	PROC rRUNSide1A200()
           	rTestPosTop;
		TPWrite "Side 1 A";
		MoveJ pSafeS1, vmax, fine, tWeldGun;
		!Code Goes Here
		MoveJ pSafeS181, vmax, fine, tWeldGun;
		SingArea\Wrist;
		MoveJ [[1181.97,1536.60,299.24],[0.0635588,0.517232,-0.779106,0.348462],[0,1,-3,1],[9E+09,9E+09,9E+09,9E+09,9E+09,9E+09]], vmax, z10, tWeldGun;
		MoveL [[1181.96,1536.60,-12.62],[0.0635661,0.517237,-0.779104,0.348458],[0,1,-2,1],[9E+09,9E+09,9E+09,9E+09,9E+09,9E+09]], v1000, z10, tWeldGun;
		ArcLStart [[1181.53,1528.23,-13.21],[0.063566,0.517241,-0.779104,0.348451],[0,1,-2,1],[9E+09,9E+09,9E+09,9E+09,9E+09,9E+09]], v10, seam13, weld13\Weave:=weave1, fine, tWeldGun;
		ArcLEnd [[1204.96,1528.67,-13.35],[0.0635597,0.517241,-0.779099,0.348465],[0,1,-2,1],[9E+09,9E+09,9E+09,9E+09,9E+09,9E+09]], v10, seam13, weld13\Weave:=weave1, fine, tWeldGun;
		MoveL [[1204.64,1537.23,-12.62],[0.0635617,0.517239,-0.7791,0.348464],[0,1,-2,1],[9E+09,9E+09,9E+09,9E+09,9E+09,9E+09]], vmax, z10, tWeldGun;
		MoveL [[863.66,1538.85,77.89],[0.0635666,0.517243,-0.779097,0.348464],[0,1,-2,1],[9E+09,9E+09,9E+09,9E+09,9E+09,9E+09]], vmax, z10, tWeldGun;
		MoveJ [[861.58,1461.21,260.09],[0.14949,-0.376148,-0.839997,-0.361347],[0,1,-1,1],[9E+09,9E+09,9E+09,9E+09,9E+09,9E+09]], vmax, z10, tWeldGun;
		MoveL [[863.23,1471.68,-11.89],[0.149517,-0.37621,-0.839967,-0.361342],[0,1,-1,1],[9E+09,9E+09,9E+09,9E+09,9E+09,9E+09]], v1000, z10, tWeldGun;
		ArcLStart [[868.03,1476.60,-13.62],[0.103036,-0.394927,-0.849321,-0.334768],[0,1,-1,1],[9E+09,9E+09,9E+09,9E+09,9E+09,9E+09]], v10, seam13, weld13\Weave:=weave1, fine, tWeldGun;
		ArcLEnd [[889.84,1476.38,-13.62],[0.103038,-0.394927,-0.849321,-0.334769],[0,1,-1,1],[9E+09,9E+09,9E+09,9E+09,9E+09,9E+09]], v10, seam13, weld13\Weave:=weave1, fine, tWeldGun;
		MoveL [[886.08,1463.03,-7.28],[0.149478,-0.376156,-0.840008,-0.361317],[0,1,-1,1],[9E+09,9E+09,9E+09,9E+09,9E+09,9E+09]], vmax, z10, tWeldGun;
		MoveJ [[863.35,1506.96,224.59],[0.0635605,0.517248,-0.779091,0.348471],[0,1,-2,1],[9E+09,9E+09,9E+09,9E+09,9E+09,9E+09]], vmax, z10, tWeldGun;
		MoveL [[863.21,1535.55,-10.64],[0.0635626,0.51725,-0.779093,0.348463],[0,1,-2,1],[9E+09,9E+09,9E+09,9E+09,9E+09,9E+09]], vmax, z10, tWeldGun;
		ArcLStart [[862.97,1528.60,-12.53],[0.0386315,0.528138,-0.780724,0.331736],[0,1,-2,1],[9E+09,9E+09,9E+09,9E+09,9E+09,9E+09]], v10, seam13, weld13\Weave:=weave1, fine, tWeldGun;
		ArcLEnd [[883.17,1528.60,-12.53],[0.0386327,0.528141,-0.780723,0.331734],[0,1,-2,1],[9E+09,9E+09,9E+09,9E+09,9E+09,9E+09]], v10, seam13, weld13\Weave:=weave1, fine, tWeldGun;
		MoveL [[887.77,1539.90,182.89],[0.0635615,0.517251,-0.779088,0.348474],[0,1,-2,1],[9E+09,9E+09,9E+09,9E+09,9E+09,9E+09]], vmax, z10, tWeldGun;
		MoveJ [[1182.52,1470.34,61.27],[0.149538,-0.376243,-0.839941,-0.361358],[0,1,-1,1],[9E+09,9E+09,9E+09,9E+09,9E+09,9E+09]], vmax, z10, tWeldGun;
		MoveL [[1182.53,1470.34,-13.67],[0.149532,-0.376236,-0.839946,-0.361356],[0,1,-1,1],[9E+09,9E+09,9E+09,9E+09,9E+09,9E+09]], v1000, z10, tWeldGun;
		ArcLStart [[1181.98,1475.51,-14.31],[0.12127,-0.382205,-0.84735,-0.348153],[0,1,-1,1],[9E+09,9E+09,9E+09,9E+09,9E+09,9E+09]], v10, seam13, weld13\Weave:=weave1, fine, tWeldGun;
		ArcLEnd [[1205.98,1475.52,-14.31],[0.121276,-0.382215,-0.847342,-0.348161],[0,1,-1,1],[9E+09,9E+09,9E+09,9E+09,9E+09,9E+09]], v10, seam13, weld13\Weave:=weave1, fine, tWeldGun;
		MoveL [[1202.33,1469.98,-15.09],[0.149549,-0.376274,-0.839922,-0.361365],[0,1,-1,1],[9E+09,9E+09,9E+09,9E+09,9E+09,9E+09]], vmax, z10, tWeldGun;
		MoveL [[1203.94,921.98,77.52],[0.149416,-0.376356,-0.839957,-0.361252],[0,1,-1,1],[9E+09,9E+09,9E+09,9E+09,9E+09,9E+09]], vmax, z10, tWeldGun;
		MoveL [[1203.94,921.99,-12.57],[0.149422,-0.37636,-0.83995,-0.361263],[0,1,-1,1],[9E+09,9E+09,9E+09,9E+09,9E+09,9E+09]], v1000, z10, tWeldGun;
		ArcLStart [[1203.92,927.58,-13.22],[0.10136,-0.39649,-0.845914,-0.341982],[0,1,-1,1],[9E+09,9E+09,9E+09,9E+09,9E+09,9E+09]], v10, seam13, weld13\Weave:=weave1, fine, tWeldGun;
		ArcLEnd [[1182.52,927.58,-13.22],[0.101362,-0.396499,-0.845908,-0.341986],[0,1,-1,1],[9E+09,9E+09,9E+09,9E+09,9E+09,9E+09]], v10, seam13, weld13\Weave:=weave1, fine, tWeldGun;
		MoveL [[1177.78,921.50,-1.65],[0.149422,-0.376364,-0.839949,-0.36126],[0,1,-1,1],[9E+09,9E+09,9E+09,9E+09,9E+09,9E+09]], vmax, z10, tWeldGun;
		MoveL [[883.71,921.14,-1.64],[0.149424,-0.37639,-0.839933,-0.361269],[0,1,0,1],[9E+09,9E+09,9E+09,9E+09,9E+09,9E+09]], vmax, z10, tWeldGun;
		MoveL [[883.71,924.70,-6.65],[0.151492,-0.376355,-0.855909,-0.320669],[0,1,-1,1],[9E+09,9E+09,9E+09,9E+09,9E+09,9E+09]], v1000, z10, tWeldGun;
		ArcLStart [[883.71,929.31,-12.65],[0.151491,-0.376316,-0.85593,-0.320657],[0,1,-1,1],[9E+09,9E+09,9E+09,9E+09,9E+09,9E+09]], v10, seam13, weld13\Weave:=weave1, fine, tWeldGun;
		ArcLEnd [[865.11,929.31,-12.65],[0.151488,-0.376316,-0.855931,-0.320655],[0,1,-1,1],[9E+09,9E+09,9E+09,9E+09,9E+09,9E+09]], v10, seam13, weld13\Weave:=weave1, fine, tWeldGun;
		MoveL [[863.70,926.54,-9.64],[0.149437,-0.376438,-0.8399,-0.361292],[0,0,0,1],[9E+09,9E+09,9E+09,9E+09,9E+09,9E+09]], v100, z10, tWeldGun;
		MoveL [[861.26,919.79,117.88],[0.149443,-0.376442,-0.8399,-0.361285],[0,1,-1,1],[9E+09,9E+09,9E+09,9E+09,9E+09,9E+09]], vmax, z0, tWeldGun;
		MoveJ [[868.17,991.07,127.71],[0.0426372,-0.330552,0.858067,-0.39069],[0,1,-2,1],[9E+09,9E+09,9E+09,9E+09,9E+09,9E+09]], vmax, z0, tWeldGun;
		MoveL [[868.52,984.75,-7.25],[0.0429876,-0.330645,0.857998,-0.390725],[0,0,-2,1],[9E+09,9E+09,9E+09,9E+09,9E+09,9E+09]], v1000, z10, tWeldGun;
		ArcLStart [[865.93,978.35,-9.72],[0.0443365,-0.337733,0.871616,-0.352502],[0,0,-1,1],[9E+09,9E+09,9E+09,9E+09,9E+09,9E+09]], v10, seam13, weld13\Weave:=weave1, fine, tWeldGun;
		ArcLEnd [[890.71,978.29,-9.75],[0.0443001,-0.337695,0.871633,-0.3525],[0,0,-1,1],[9E+09,9E+09,9E+09,9E+09,9E+09,9E+09]], v10, seam13, weld13\Weave:=weave1, fine, tWeldGun;
		MoveL [[889.59,992.71,-6.61],[0.0430178,-0.330607,0.858002,-0.390745],[0,0,-2,1],[9E+09,9E+09,9E+09,9E+09,9E+09,9E+09]], vmax, z10, tWeldGun;
		MoveL [[889.59,992.73,75.52],[0.0430306,-0.330621,0.857997,-0.390743],[0,1,-2,1],[9E+09,9E+09,9E+09,9E+09,9E+09,9E+09]], vmax, z10, tWeldGun;
		MoveL [[1177.66,992.72,75.52],[0.0430182,-0.33062,0.857997,-0.390745],[0,0,-2,1],[9E+09,9E+09,9E+09,9E+09,9E+09,9E+09]], vmax, z10, tWeldGun;
		MoveL [[1185.40,982.49,-9.15],[0.0429596,-0.330615,0.858003,-0.390743],[0,0,-2,1],[9E+09,9E+09,9E+09,9E+09,9E+09,9E+09]], v1000, z10, tWeldGun;
		ArcLStart [[1180.06,977.10,-12.03],[0.0429555,-0.330634,0.857992,-0.390751],[0,0,-2,1],[9E+09,9E+09,9E+09,9E+09,9E+09,9E+09]], v10, seam13, weld13\Weave:=weave1, fine, tWeldGun;
		ArcLEnd [[1208.25,977.44,-12.05],[0.0429485,-0.330644,0.85799,-0.390748],[0,0,-2,1],[9E+09,9E+09,9E+09,9E+09,9E+09,9E+09]], v10, seam13, weld13\Weave:=weave1, fine, tWeldGun;
		MoveL [[1207.94,989.04,-11.16],[0.0429397,-0.330625,0.858002,-0.39074],[0,0,-2,1],[9E+09,9E+09,9E+09,9E+09,9E+09,9E+09]], v1000, z10, tWeldGun;
		MoveL [[1207.95,989.04,392.36],[0.0429563,-0.330627,0.857995,-0.39075],[0,1,-2,1],[9E+09,9E+09,9E+09,9E+09,9E+09,9E+09]], vmax, z10, tWeldGun;
		MoveJ [[194.09,1536.38,108.42],[0.0907205,-0.623393,0.712906,0.308084],[0,-1,0,1],[9E+09,9E+09,9E+09,9E+09,9E+09,9E+09]], vmax, z10, tWeldGun;
		MoveL [[194.09,1534.55,44.51],[0.0907126,-0.623398,0.712901,0.308089],[0,-1,0,1],[9E+09,9E+09,9E+09,9E+09,9E+09,9E+09]], vmax, z10, tWeldGun;
		ArcLStart [[188.67,1534.52,-1.78],[0.0904696,-0.623399,0.71298,0.307975],[0,-1,0,1],[9E+09,9E+09,9E+09,9E+09,9E+09,9E+09]], v20, seam13, weld13\Weave:=weave1, fine, tWeldGun;
		ArcLEnd [[157.07,1534.50,-1.61],[0.0904549,-0.623403,0.712983,0.307965],[0,-1,0,1],[9E+09,9E+09,9E+09,9E+09,9E+09,9E+09]], v20, seam13, weld13\Weave:=weave1, fine, tWeldGun;
		MoveL [[158.09,1532.35,8.43],[0.0907075,-0.623402,0.712898,0.30809],[0,-1,0,1],[9E+09,9E+09,9E+09,9E+09,9E+09,9E+09]], vmax, z10, tWeldGun;
		MoveL [[-123.91,1535.35,12.43],[0.0907124,-0.623396,0.712903,0.308089],[1,0,0,1],[9E+09,9E+09,9E+09,9E+09,9E+09,9E+09]], vmax, z10, tWeldGun;
		ArcLStart [[-128.10,1535.33,-0.77],[0.0907065,-0.623392,0.712906,0.308093],[1,0,0,1],[9E+09,9E+09,9E+09,9E+09,9E+09,9E+09]], v20, seam13, weld13\Weave:=weave1, fine, tWeldGun;
		ArcLEnd [[-161.33,1535.32,-0.76],[0.0907026,-0.623409,0.712891,0.308093],[1,0,0,1],[9E+09,9E+09,9E+09,9E+09,9E+09,9E+09]], v20, seam13, weld13\Weave:=weave1, fine, tWeldGun;
		MoveL [[-158.90,1535.32,931.69],[0.0906389,-0.623348,0.712932,0.308139],[1,-2,1,0],[9E+09,9E+09,9E+09,9E+09,9E+09,9E+09]], vmax, z0, tWeldGun;
		MoveJ [[-173.66,614.72,251.09],[0.128906,0.0495871,0.95885,-0.248055],[1,-1,1,0],[9E+09,9E+09,9E+09,9E+09,9E+09,9E+09]], vmax, z0, tWeldGun;
		MoveL [[-146.66,553.40,15.33],[0.15216,0.0393582,0.96563,-0.207021],[1,-1,1,0],[9E+09,9E+09,9E+09,9E+09,9E+09,9E+09]], vmax, z0, tWeldGun;
		ArcLStart [[-147.88,553.18,1.12],[0.150717,0.044516,0.958032,-0.239748],[1,-1,1,0],[9E+09,9E+09,9E+09,9E+09,9E+09,9E+09]], v20, seam13, weld13\Weave:=weave1, fine, tWeldGun;
		ArcLEnd [[-115.28,553.19,1.13],[0.150723,0.044502,0.958032,-0.239744],[1,-1,1,0],[9E+09,9E+09,9E+09,9E+09,9E+09,9E+09]], v20, seam13, weld13\Weave:=weave1, fine, tWeldGun;
		MoveL [[-113.65,555.41,12.33],[0.152159,0.0393397,0.96563,-0.207027],[1,-1,1,0],[9E+09,9E+09,9E+09,9E+09,9E+09,9E+09]], vmax, z0, tWeldGun;
		MoveL [[171.61,552.68,21.42],[0.152083,0.0394694,0.965633,-0.207041],[1,-1,1,0],[9E+09,9E+09,9E+09,9E+09,9E+09,9E+09]], vmax, z0, tWeldGun;
		ArcLStart [[168.61,552.48,-0.51],[0.15096,0.043697,0.959444,-0.234031],[1,-1,1,0],[9E+09,9E+09,9E+09,9E+09,9E+09,9E+09]], v20, seam13, weld13\Weave:=weave1, fine, tWeldGun;
		ArcLEnd [[200.42,552.49,-0.51],[0.150963,0.0436867,0.959444,-0.23403],[1,-1,1,0],[9E+09,9E+09,9E+09,9E+09,9E+09,9E+09]], v20, seam13, weld13\Weave:=weave1, fine, tWeldGun;
		MoveL [[204.25,552.75,13.91],[0.152145,0.0394344,0.965619,-0.207068],[1,-1,1,0],[9E+09,9E+09,9E+09,9E+09,9E+09,9E+09]], vmax, z0, tWeldGun;
		MoveL [[860.18,549.11,14.83],[0.152112,0.039289,0.965636,-0.207043],[0,-2,1,0],[9E+09,9E+09,9E+09,9E+09,9E+09,9E+09]], vmax, z0, tWeldGun;
		ArcLStart [[862.38,548.31,-2.96],[0.133579,0.0504356,0.95444,-0.262026],[0,-1,1,0],[9E+09,9E+09,9E+09,9E+09,9E+09,9E+09]], v20, seam13, weld13\Weave:=weave1, fine, tWeldGun;
		ArcLEnd [[895.35,548.90,-2.97],[0.133556,0.0504648,0.954436,-0.262046],[0,-2,1,0],[9E+09,9E+09,9E+09,9E+09,9E+09,9E+09]], v20, seam13, weld13\Weave:=weave1, fine, tWeldGun;
		MoveL [[895.37,549.34,9.83],[0.15211,0.0392827,0.965635,-0.207047],[0,-2,1,0],[9E+09,9E+09,9E+09,9E+09,9E+09,9E+09]], vmax, z0, tWeldGun;
		MoveL [[1175.32,546.94,11.83],[0.1496,0.0478929,0.95235,-0.261449],[0,-2,1,0],[9E+09,9E+09,9E+09,9E+09,9E+09,9E+09]], vmax, z0, tWeldGun;
		ArcLStart [[1179.08,546.13,-3.58],[0.119147,0.061512,0.947538,-0.290161],[0,-2,1,0],[9E+09,9E+09,9E+09,9E+09,9E+09,9E+09]], v20, seam13, weld13\Weave:=weave1, fine, tWeldGun;
		ArcLEnd [[1209.46,546.13,-3.60],[0.15155,0.0512739,0.944084,-0.288288],[0,-2,1,0],[9E+09,9E+09,9E+09,9E+09,9E+09,9E+09]], v20, seam13, weld13\Weave:=weave1, fine, tWeldGun;
		MoveL [[1183.76,537.75,320.86],[0.152128,0.0394118,0.965637,-0.207003],[0,-2,1,0],[9E+09,9E+09,9E+09,9E+09,9E+09,9E+09]], vmax, z0, tWeldGun;
		MoveJ [[759.22,820.77,477.02],[0.128857,0.0495447,0.958803,-0.24827],[0,-1,1,0],[9E+09,9E+09,9E+09,9E+09,9E+09,9E+09]], vmax, z0, tWeldGun;
		MoveJ [[-401.88,982.38,420.80],[0.377905,-0.177501,-0.908663,-0.00353082],[1,0,1,0],[9E+09,9E+09,9E+09,9E+09,9E+09,9E+09]], vmax, z0, tWeldGun;
		MoveL [[-401.87,982.37,-5.96],[0.377901,-0.177501,-0.908665,-0.00352363],[1,0,1,0],[9E+09,9E+09,9E+09,9E+09,9E+09,9E+09]], v1000, z0, tWeldGun;
		ArcLStart [[-407.78,982.54,-7.55],[0.377944,-0.177367,-0.908673,-0.00361758],[1,0,1,0],[9E+09,9E+09,9E+09,9E+09,9E+09,9E+09]], v10, seam13, weld13\Weave:=weave1, fine, tWeldGun;
		ArcL [[-407.62,961.97,-9.33],[0.377925,-0.177522,-0.908651,-0.00352087],[1,0,1,0],[9E+09,9E+09,9E+09,9E+09,9E+09,9E+09]], v10, seam13, weld13\Weave:=weave1, z10, tWeldGun;
		ArcLEnd [[-429.63,955.24,-8.57],[0.245864,-0.589236,-0.75089,-0.168871],[1,0,2,0],[9E+09,9E+09,9E+09,9E+09,9E+09,9E+09]], v10, seam13, weld13\Weave:=weave1, fine, tWeldGun;
		MoveL [[-432.47,945.01,-6.78],[0.274937,-0.581449,-0.743579,-0.182803],[1,0,2,0],[9E+09,9E+09,9E+09,9E+09,9E+09,9E+09]], vmax, z0, tWeldGun;
		MoveL [[-432.39,895.03,94.24],[0.274951,-0.581467,-0.743558,-0.182811],[1,0,2,0],[9E+09,9E+09,9E+09,9E+09,9E+09,9E+09]], vmax, z0, tWeldGun;
		MoveL [[-1101.20,895.02,94.24],[0.274939,-0.581469,-0.743563,-0.182805],[1,0,2,0],[9E+09,9E+09,9E+09,9E+09,9E+09,9E+09]], vmax, z0, tWeldGun;
		MoveL [[-1101.70,938.01,-1.40],[0.240452,-0.654006,-0.686015,-0.209388],[1,0,2,0],[9E+09,9E+09,9E+09,9E+09,9E+09,9E+09]], v1000, z0, tWeldGun;
		ArcLStart [[-1101.62,952.01,-7.20],[0.240453,-0.653997,-0.686023,-0.209388],[1,0,2,0],[9E+09,9E+09,9E+09,9E+09,9E+09,9E+09]], v10, seam13, weld13\Weave:=weave1, fine, tWeldGun;
		ArcL [[-1123.02,952.13,-5.59],[0.240455,-0.654006,-0.686013,-0.209388],[1,0,2,0],[9E+09,9E+09,9E+09,9E+09,9E+09,9E+09]], v10, seam13, weld13\Weave:=weave1, z10, tWeldGun;
		ArcLEnd [[-1128.50,976.05,-6.40],[0.0369824,0.922972,0.0835342,0.37387],[1,0,3,0],[9E+09,9E+09,9E+09,9E+09,9E+09,9E+09]], v10, seam13, weld13\Weave:=weave1, fine, tWeldGun;
		MoveL [[-1142.99,977.01,6.44],[0.0501214,0.923455,0.0523108,0.376805],[1,0,3,0],[9E+09,9E+09,9E+09,9E+09,9E+09,9E+09]], vmax, z0, tWeldGun;
		MoveJ [[-1224.84,979.29,303.50],[0.0444685,0.923113,0.0666376,0.376092],[1,0,-1,0],[9E+09,9E+09,9E+09,9E+09,9E+09,9E+09]], vmax, z20, tWeldGun;
		MoveL [[-1192.76,1156.53,-4.42],[0.044443,0.923122,0.0666432,0.376072],[1,0,-1,0],[9E+09,9E+09,9E+09,9E+09,9E+09,9E+09]], v1000, z0, tWeldGun;
		ArcLStart [[-1191.66,1156.15,-2.46],[0.0444485,0.92313,0.0666399,0.376052],[1,0,-1,0],[9E+09,9E+09,9E+09,9E+09,9E+09,9E+09]], v10, seam13, weld13\Weave:=weave1, fine, tWeldGun;
		ArcL [[-1191.78,1180.21,-3.92],[0.0444409,0.923134,0.066615,0.376047],[1,0,-1,0],[9E+09,9E+09,9E+09,9E+09,9E+09,9E+09]], v10, seam13, weld13\Weave:=weave1, z10, tWeldGun;
		ArcLEnd [[-1166.74,1189.82,-5.14],[0.269841,0.674631,-0.631942,0.269645],[1,0,0,0],[9E+09,9E+09,9E+09,9E+09,9E+09,9E+09]], v10, seam13, weld13\Weave:=weave1, fine, tWeldGun;
		MoveL [[-1165.81,1197.81,-4.44],[0.289046,0.665942,-0.622199,0.292988],[1,0,0,0],[9E+09,9E+09,9E+09,9E+09,9E+09,9E+09]], vmax, z0, tWeldGun;
		MoveL [[-1167.37,1197.80,267.48],[0.269054,0.631082,-0.684208,0.247398],[1,-1,0,0],[9E+09,9E+09,9E+09,9E+09,9E+09,9E+09]], vmax, z0, tWeldGun;
		MoveJ [[-491.85,1197.38,267.48],[0.269045,0.631086,-0.684208,0.247399],[1,-1,0,0],[9E+09,9E+09,9E+09,9E+09,9E+09,9E+09]], vmax, z0, tWeldGun;
		MoveL [[-493.75,1206.46,4.64],[0.230361,0.671978,-0.666396,0.226485],[1,-1,0,0],[9E+09,9E+09,9E+09,9E+09,9E+09,9E+09]], v1000, z0, tWeldGun;
		ArcLStart [[-493.89,1194.98,-8.68],[0.230347,0.671983,-0.666395,0.226488],[1,-1,0,0],[9E+09,9E+09,9E+09,9E+09,9E+09,9E+09]], v10, seam13, weld13\Weave:=weave1, fine, tWeldGun;
		ArcL [[-474.80,1194.46,-8.19],[0.230358,0.671985,-0.666393,0.22648],[1,-1,0,0],[9E+09,9E+09,9E+09,9E+09,9E+09,9E+09]], v10, seam13, weld13\Weave:=weave1, z10, tWeldGun;
		ArcLEnd [[-467.21,1164.88,-9.76],[0.384925,0.00804859,-0.922637,-0.0225884],[1,-1,1,0],[9E+09,9E+09,9E+09,9E+09,9E+09,9E+09]], v10, seam13, weld13\Weave:=weave1, fine, tWeldGun;
		MoveL [[-460.21,1166.10,-6.29],[0.384934,0.00803439,-0.922633,-0.0226006],[1,-1,1,0],[9E+09,9E+09,9E+09,9E+09,9E+09,9E+09]], vmax, z5, tWeldGun;
		MoveL [[-460.61,1166.13,158.38],[0.384913,0.00804793,-0.922641,-0.0226089],[1,-1,1,0],[9E+09,9E+09,9E+09,9E+09,9E+09,9E+09]], vmax, z5, tWeldGun;
		MoveJ [[-411.67,714.00,66.77],[0.262804,0.646065,-0.670013,0.254199],[1,-1,0,0],[9E+09,9E+09,9E+09,9E+09,9E+09,9E+09]], vmax, z5, tWeldGun;
		MoveL [[-411.69,717.21,-6.09],[0.256237,0.656032,-0.660062,0.261312],[1,-1,0,0],[9E+09,9E+09,9E+09,9E+09,9E+09,9E+09]], vmax, z5, tWeldGun;
		ArcLStart [[-411.68,712.41,-5.70],[0.256247,0.656027,-0.66006,0.261318],[1,-1,0,0],[9E+09,9E+09,9E+09,9E+09,9E+09,9E+09]], v5, seam13, weld13\Weave:=weave1, fine, tWeldGun;
		ArcLEnd [[-433.47,712.42,-5.71],[0.256245,0.656034,-0.660051,0.261328],[1,-1,0,0],[9E+09,9E+09,9E+09,9E+09,9E+09,9E+09]], v5, seam13, weld13\Weave:=weave1, fine, tWeldGun;
		MoveL [[-433.52,712.50,86.63],[0.256209,0.656106,-0.660016,0.261269],[1,-1,0,0],[9E+09,9E+09,9E+09,9E+09,9E+09,9E+09]], vmax, z5, tWeldGun;
		MoveL [[-1103.37,713.70,123.92],[0.256219,0.656103,-0.660014,0.261271],[1,-1,0,0],[9E+09,9E+09,9E+09,9E+09,9E+09,9E+09]], vmax, z5, tWeldGun;
		MoveL [[-1103.36,713.70,-5.85],[0.25622,0.656101,-0.660014,0.261276],[1,-1,0,0],[9E+09,9E+09,9E+09,9E+09,9E+09,9E+09]], vmax, z5, tWeldGun;
		ArcLStart [[-1100.80,710.80,-5.85],[0.25621,0.656115,-0.660005,0.261274],[1,-1,0,0],[9E+09,9E+09,9E+09,9E+09,9E+09,9E+09]], v5, seam13, weld13\Weave:=weave1, fine, tWeldGun;
		ArcLEnd [[-1124.56,710.81,-5.88],[0.256211,0.6561,-0.660011,0.261294],[1,-1,0,0],[9E+09,9E+09,9E+09,9E+09,9E+09,9E+09]], v5, seam13, weld13\Weave:=weave1, fine, tWeldGun;
		MoveL [[-1124.57,723.78,145.38],[0.256225,0.656093,-0.660015,0.261287],[1,-1,0,0],[9E+09,9E+09,9E+09,9E+09,9E+09,9E+09]], vmax, z5, tWeldGun;
		MoveJ [[-1174.22,1417.20,153.64],[0.288404,-0.63354,-0.657568,-0.288193],[1,-1,-2,0],[9E+09,9E+09,9E+09,9E+09,9E+09,9E+09]], vmax, z5, tWeldGun;
		MoveL [[-1186.57,1426.06,2.31],[0.28839,-0.633552,-0.657559,-0.288201],[1,-1,-2,0],[9E+09,9E+09,9E+09,9E+09,9E+09,9E+09]], vmax, z5, tWeldGun;
		ArcLStart [[-1185.81,1430.45,-4.51],[0.288383,-0.633572,-0.657547,-0.288192],[1,-1,-2,0],[9E+09,9E+09,9E+09,9E+09,9E+09,9E+09]], v5, seam13, weld13\Weave:=weave1, fine, tWeldGun;
		ArcLEnd [[-1165.69,1430.23,-5.50],[0.288385,-0.633579,-0.65754,-0.288189],[1,-1,-2,0],[9E+09,9E+09,9E+09,9E+09,9E+09,9E+09]], v5, seam13, weld13\Weave:=weave1, fine, tWeldGun;
		MoveL [[-1165.69,1421.27,86.72],[0.28839,-0.633573,-0.657541,-0.288197],[1,-1,-2,0],[9E+09,9E+09,9E+09,9E+09,9E+09,9E+09]], vmax, z5, tWeldGun;
		MoveL [[-494.06,1426.01,134.66],[0.280642,-0.634844,-0.656104,-0.296212],[1,-1,-2,0],[9E+09,9E+09,9E+09,9E+09,9E+09,9E+09]], vmax, z5, tWeldGun;
		MoveL [[-494.05,1425.99,-2.61],[0.280635,-0.634843,-0.65611,-0.296207],[1,-1,-2,0],[9E+09,9E+09,9E+09,9E+09,9E+09,9E+09]], vmax, z5, tWeldGun;
		ArcLStart [[-494.25,1431.59,-10.43],[0.280631,-0.634852,-0.656104,-0.296205],[1,-1,-2,0],[9E+09,9E+09,9E+09,9E+09,9E+09,9E+09]], v5, seam13, weld13\Weave:=weave1, fine, tWeldGun;
		ArcLEnd [[-471.85,1431.77,-9.45],[0.280622,-0.634875,-0.656087,-0.296202],[1,-1,-2,0],[9E+09,9E+09,9E+09,9E+09,9E+09,9E+09]], v5, seam13, weld13\Weave:=weave1, fine, tWeldGun;
		MoveL [[-471.84,1418.41,452.48],[0.280608,-0.634847,-0.656147,-0.296143],[1,-1,-2,0],[9E+09,9E+09,9E+09,9E+09,9E+09,9E+09]], vmax, z5, tWeldGun;
		MoveJ pSafeS1, vmax, fine, tWeldGun;
	ENDPROC
	PROC ss_200()
           	rTestPosTop;
		TPWrite "Side 1 A";
		MoveJ pSafeS1, vmax, fine, tWeldGun;
		!Code Goes Here
		MoveJ pSafeS181, vmax, fine, tWeldGun;
		SingArea\Wrist;
		MoveJ [[1181.97,1536.60,299.24],[0.0635588,0.517232,-0.779106,0.348462],[0,1,-3,1],[9E+09,9E+09,9E+09,9E+09,9E+09,9E+09]], vmax, z10, tWeldGun;
		MoveL [[1181.96,1536.60,-12.62],[0.0635661,0.517237,-0.779104,0.348458],[0,1,-2,1],[9E+09,9E+09,9E+09,9E+09,9E+09,9E+09]], v1000, z10, tWeldGun;
		ArcLStart [[1181.53,1529.02,-11.65],[0.0635714,0.517237,-0.779104,0.348457],[0,1,-2,1],[9E+09,9E+09,9E+09,9E+09,9E+09,9E+09]], v10, seam13, weld13\Weave:=weave1, fine, tWeldGun;
		ArcLEnd [[1204.96,1529.87,-10.62],[0.0635614,0.517237,-0.779103,0.348461],[0,1,-2,1],[9E+09,9E+09,9E+09,9E+09,9E+09,9E+09]], v10, seam13, weld13\Weave:=weave1, fine, tWeldGun;
		MoveL [[1204.64,1537.23,-12.62],[0.0635617,0.517239,-0.7791,0.348464],[0,1,-2,1],[9E+09,9E+09,9E+09,9E+09,9E+09,9E+09]], vmax, z10, tWeldGun;
		MoveL [[863.66,1538.85,77.89],[0.0635666,0.517243,-0.779097,0.348464],[0,1,-2,1],[9E+09,9E+09,9E+09,9E+09,9E+09,9E+09]], vmax, z10, tWeldGun;
		MoveJ [[861.58,1461.21,260.09],[0.14949,-0.376148,-0.839997,-0.361347],[0,1,-1,1],[9E+09,9E+09,9E+09,9E+09,9E+09,9E+09]], vmax, z10, tWeldGun;
		MoveL [[863.23,1471.68,-11.89],[0.149517,-0.37621,-0.839967,-0.361342],[0,1,-1,1],[9E+09,9E+09,9E+09,9E+09,9E+09,9E+09]], v1000, z10, tWeldGun;
		ArcLStart [[863.88,1474.96,-12.64],[0.149558,-0.376296,-0.839897,-0.361396],[0,1,-1,1],[9E+09,9E+09,9E+09,9E+09,9E+09,9E+09]], v10, seam13, weld13\Weave:=weave1, fine, tWeldGun;
		ArcLEnd [[887.67,1475.21,-13.25],[0.149548,-0.376266,-0.839942,-0.361327],[0,1,-1,1],[9E+09,9E+09,9E+09,9E+09,9E+09,9E+09]], v10, seam13, weld13\Weave:=weave1, fine, tWeldGun;
		MoveL [[886.08,1463.03,-7.28],[0.149478,-0.376156,-0.840008,-0.361317],[0,1,-1,1],[9E+09,9E+09,9E+09,9E+09,9E+09,9E+09]], vmax, z10, tWeldGun;
		MoveJ [[863.35,1506.96,224.59],[0.0635605,0.517248,-0.779091,0.348471],[0,1,-2,1],[9E+09,9E+09,9E+09,9E+09,9E+09,9E+09]], vmax, z10, tWeldGun;
		MoveL [[863.21,1535.55,-10.64],[0.0635626,0.51725,-0.779093,0.348463],[0,1,-2,1],[9E+09,9E+09,9E+09,9E+09,9E+09,9E+09]], vmax, z10, tWeldGun;
		ArcLStart [[862.98,1531.20,-11.14],[0.0635851,0.517245,-0.779094,0.348464],[0,1,-2,1],[9E+09,9E+09,9E+09,9E+09,9E+09,9E+09]], v10, seam13, weld13\Weave:=weave1, fine, tWeldGun;
		ArcLEnd [[887.38,1530.81,-10.94],[0.0635922,0.517251,-0.779089,0.348465],[0,1,-2,1],[9E+09,9E+09,9E+09,9E+09,9E+09,9E+09]], v10, seam13, weld13\Weave:=weave1, fine, tWeldGun;
		MoveL [[887.77,1539.90,182.89],[0.0635615,0.517251,-0.779088,0.348474],[0,1,-2,1],[9E+09,9E+09,9E+09,9E+09,9E+09,9E+09]], vmax, z10, tWeldGun;
		MoveJ [[1182.52,1470.34,61.27],[0.149538,-0.376243,-0.839941,-0.361358],[0,1,-1,1],[9E+09,9E+09,9E+09,9E+09,9E+09,9E+09]], vmax, z10, tWeldGun;
		MoveL [[1182.53,1470.34,-16.07],[0.149529,-0.376231,-0.83995,-0.361353],[0,1,-1,1],[9E+09,9E+09,9E+09,9E+09,9E+09,9E+09]], v1000, z10, tWeldGun;
		ArcLStart [[1181.99,1475.51,-15.52],[0.149552,-0.376279,-0.83992,-0.361363],[0,1,-1,1],[9E+09,9E+09,9E+09,9E+09,9E+09,9E+09]], v10, seam13, weld13\Weave:=weave1, fine, tWeldGun;
		ArcLEnd [[1204.38,1476.47,-15.60],[0.149569,-0.376356,-0.839878,-0.361375],[0,1,-1,1],[9E+09,9E+09,9E+09,9E+09,9E+09,9E+09]], v10, seam13, weld13\Weave:=weave1, fine, tWeldGun;
		MoveL [[1202.33,1469.98,-15.09],[0.149549,-0.376274,-0.839922,-0.361365],[0,1,-1,1],[9E+09,9E+09,9E+09,9E+09,9E+09,9E+09]], vmax, z10, tWeldGun;
		MoveL [[1203.94,921.98,77.52],[0.149416,-0.376356,-0.839957,-0.361252],[0,1,-1,1],[9E+09,9E+09,9E+09,9E+09,9E+09,9E+09]], vmax, z10, tWeldGun;
		MoveL [[1203.94,921.99,-12.97],[0.149422,-0.376348,-0.839957,-0.361259],[0,1,-1,1],[9E+09,9E+09,9E+09,9E+09,9E+09,9E+09]], v1000, z10, tWeldGun;
		ArcLStart [[1203.94,928.79,-14.21],[0.149423,-0.376362,-0.839952,-0.361256],[0,1,-1,1],[9E+09,9E+09,9E+09,9E+09,9E+09,9E+09]], v10, seam13, weld13\Weave:=weave1, fine, tWeldGun;
		ArcLEnd [[1178.19,928.79,-14.21],[0.149422,-0.376442,-0.839904,-0.361285],[0,1,-1,1],[9E+09,9E+09,9E+09,9E+09,9E+09,9E+09]], v10, seam13, weld13\Weave:=weave1, fine, tWeldGun;
		MoveL [[1177.78,921.50,-1.65],[0.149422,-0.376364,-0.839949,-0.36126],[0,1,-1,1],[9E+09,9E+09,9E+09,9E+09,9E+09,9E+09]], vmax, z10, tWeldGun;
		MoveL [[883.71,921.14,-1.64],[0.149424,-0.37639,-0.839933,-0.361269],[0,1,0,1],[9E+09,9E+09,9E+09,9E+09,9E+09,9E+09]], vmax, z10, tWeldGun;
		MoveL [[883.71,926.93,-12.24],[0.149423,-0.3764,-0.839927,-0.361273],[0,0,0,1],[9E+09,9E+09,9E+09,9E+09,9E+09,9E+09]], v1000, z10, tWeldGun;
		ArcLStart [[885.40,928.75,-13.38],[0.149454,-0.376503,-0.839867,-0.361295],[0,0,0,1],[9E+09,9E+09,9E+09,9E+09,9E+09,9E+09]], v10, seam13, weld13\Weave:=weave1, fine, tWeldGun;
		ArcLEnd [[866.41,928.73,-13.39],[0.149444,-0.376494,-0.839881,-0.361275],[0,0,0,1],[9E+09,9E+09,9E+09,9E+09,9E+09,9E+09]], v10, seam13, weld13\Weave:=weave1, fine, tWeldGun;
		MoveL [[863.70,926.54,-12.25],[0.149435,-0.37642,-0.839913,-0.361282],[0,0,0,1],[9E+09,9E+09,9E+09,9E+09,9E+09,9E+09]], v100, z10, tWeldGun;
		MoveL [[861.26,919.79,117.88],[0.149443,-0.376442,-0.8399,-0.361285],[0,1,-1,1],[9E+09,9E+09,9E+09,9E+09,9E+09,9E+09]], vmax, z0, tWeldGun;
		MoveJ [[868.17,991.07,127.71],[0.0426372,-0.330552,0.858067,-0.39069],[0,1,-2,1],[9E+09,9E+09,9E+09,9E+09,9E+09,9E+09]], vmax, z0, tWeldGun;
		MoveL [[868.52,991.54,-9.45],[0.0429862,-0.330642,0.857997,-0.390729],[0,0,-2,1],[9E+09,9E+09,9E+09,9E+09,9E+09,9E+09]], v1000, z10, tWeldGun;
		ArcLStart [[865.93,978.35,-10.52],[0.0429801,-0.330651,0.857991,-0.390736],[0,0,-2,1],[9E+09,9E+09,9E+09,9E+09,9E+09,9E+09]], v10, seam13, weld13\Weave:=weave1, fine, tWeldGun;
		ArcLEnd [[888.37,978.36,-11.00],[0.0429914,-0.330695,0.857973,-0.390738],[0,0,-2,1],[9E+09,9E+09,9E+09,9E+09,9E+09,9E+09]], v10, seam13, weld13\Weave:=weave1, fine, tWeldGun;
		MoveL [[889.59,992.71,-9.41],[0.0430222,-0.330607,0.858002,-0.390746],[0,0,-2,1],[9E+09,9E+09,9E+09,9E+09,9E+09,9E+09]], vmax, z10, tWeldGun;
		MoveL [[889.59,992.73,75.52],[0.0430306,-0.330621,0.857997,-0.390743],[0,1,-2,1],[9E+09,9E+09,9E+09,9E+09,9E+09,9E+09]], vmax, z10, tWeldGun;
		MoveL [[1177.66,992.72,75.52],[0.0430182,-0.33062,0.857997,-0.390745],[0,0,-2,1],[9E+09,9E+09,9E+09,9E+09,9E+09,9E+09]], vmax, z10, tWeldGun;
		MoveL [[1185.41,992.70,-11.53],[0.0429716,-0.330606,0.858007,-0.390739],[0,0,-2,1],[9E+09,9E+09,9E+09,9E+09,9E+09,9E+09]], v1000, z10, tWeldGun;
		ArcLStart [[1180.66,978.10,-13.63],[0.0429557,-0.330625,0.857997,-0.390747],[0,0,-2,1],[9E+09,9E+09,9E+09,9E+09,9E+09,9E+09]], v10, seam13, weld13\Weave:=weave1, fine, tWeldGun;
		ArcLEnd [[1207.05,977.71,-13.62],[0.0429527,-0.330628,0.857994,-0.390751],[0,0,-2,1],[9E+09,9E+09,9E+09,9E+09,9E+09,9E+09]], v10, seam13, weld13\Weave:=weave1, fine, tWeldGun;
		MoveL [[1207.94,989.04,-11.16],[0.0429397,-0.330625,0.858002,-0.39074],[0,0,-2,1],[9E+09,9E+09,9E+09,9E+09,9E+09,9E+09]], v1000, z10, tWeldGun;
		MoveL [[1207.95,989.04,392.36],[0.0429563,-0.330627,0.857995,-0.39075],[0,1,-2,1],[9E+09,9E+09,9E+09,9E+09,9E+09,9E+09]], vmax, z10, tWeldGun;
		MoveJ [[194.09,1536.38,108.42],[0.0907205,-0.623393,0.712906,0.308084],[0,-1,0,1],[9E+09,9E+09,9E+09,9E+09,9E+09,9E+09]], vmax, z10, tWeldGun;
		MoveL [[194.09,1534.55,44.51],[0.0907126,-0.623398,0.712901,0.308089],[0,-1,0,1],[9E+09,9E+09,9E+09,9E+09,9E+09,9E+09]], vmax, z10, tWeldGun;
		ArcLStart [[191.25,1532.54,0.05],[0.0904838,-0.623408,0.712969,0.30798],[0,-1,0,1],[9E+09,9E+09,9E+09,9E+09,9E+09,9E+09]], v20, seam13, weld13\Weave:=weave1, fine, tWeldGun;
		ArcLEnd [[157.22,1532.54,0.51],[0.090482,-0.623409,0.712967,0.307981],[0,-1,0,1],[9E+09,9E+09,9E+09,9E+09,9E+09,9E+09]], v20, seam13, weld13\Weave:=weave1, fine, tWeldGun;
		MoveL [[158.09,1532.35,8.43],[0.0907075,-0.623402,0.712898,0.30809],[0,-1,0,1],[9E+09,9E+09,9E+09,9E+09,9E+09,9E+09]], vmax, z10, tWeldGun;
		MoveL [[-123.91,1535.35,12.43],[0.0907124,-0.623396,0.712903,0.308089],[1,0,0,1],[9E+09,9E+09,9E+09,9E+09,9E+09,9E+09]], vmax, z10, tWeldGun;
		ArcLStart [[-126.92,1534.33,1.43],[0.0907044,-0.623405,0.712895,0.308091],[1,0,0,1],[9E+09,9E+09,9E+09,9E+09,9E+09,9E+09]], v20, seam13, weld13\Weave:=weave1, fine, tWeldGun;
		ArcLEnd [[-160.92,1534.33,1.44],[0.090708,-0.623403,0.712896,0.308092],[1,0,0,1],[9E+09,9E+09,9E+09,9E+09,9E+09,9E+09]], v20, seam13, weld13\Weave:=weave1, fine, tWeldGun;
		MoveL [[-158.90,1535.32,931.69],[0.0906389,-0.623348,0.712932,0.308139],[1,-2,1,0],[9E+09,9E+09,9E+09,9E+09,9E+09,9E+09]], vmax, z0, tWeldGun;
		MoveJ [[-173.66,614.72,251.09],[0.128906,0.0495871,0.95885,-0.248055],[1,-1,1,0],[9E+09,9E+09,9E+09,9E+09,9E+09,9E+09]], vmax, z0, tWeldGun;
		MoveL [[-146.66,553.40,15.33],[0.15216,0.0393582,0.96563,-0.207021],[1,-1,1,0],[9E+09,9E+09,9E+09,9E+09,9E+09,9E+09]], vmax, z0, tWeldGun;
		ArcLStart [[-146.66,553.39,2.32],[0.152156,0.0393511,0.965628,-0.207036],[1,-1,1,0],[9E+09,9E+09,9E+09,9E+09,9E+09,9E+09]], v20, seam13, weld13\Weave:=weave1, fine, tWeldGun;
		ArcLEnd [[-114.67,554.39,1.31],[0.152148,0.0393507,0.965628,-0.207043],[1,-1,1,0],[9E+09,9E+09,9E+09,9E+09,9E+09,9E+09]], v20, seam13, weld13\Weave:=weave1, fine, tWeldGun;
		MoveL [[-113.65,555.41,12.33],[0.152159,0.0393397,0.96563,-0.207027],[1,-1,1,0],[9E+09,9E+09,9E+09,9E+09,9E+09,9E+09]], vmax, z0, tWeldGun;
		MoveL [[171.61,552.68,21.42],[0.152083,0.0394694,0.965633,-0.207041],[1,-1,1,0],[9E+09,9E+09,9E+09,9E+09,9E+09,9E+09]], vmax, z0, tWeldGun;
		ArcLStart [[171.63,552.69,-0.51],[0.152132,0.0394445,0.96562,-0.207073],[1,-1,1,0],[9E+09,9E+09,9E+09,9E+09,9E+09,9E+09]], v20, seam13, weld13\Weave:=weave1, fine, tWeldGun;
		ArcLEnd [[202.63,552.69,-0.52],[0.152129,0.0394303,0.965618,-0.207083],[1,-1,1,0],[9E+09,9E+09,9E+09,9E+09,9E+09,9E+09]], v20, seam13, weld13\Weave:=weave1, fine, tWeldGun;
		MoveL [[204.25,552.75,13.91],[0.152145,0.0394344,0.965619,-0.207068],[1,-1,1,0],[9E+09,9E+09,9E+09,9E+09,9E+09,9E+09]], vmax, z0, tWeldGun;
		MoveL [[860.18,549.11,14.83],[0.152112,0.039289,0.965636,-0.207043],[0,-2,1,0],[9E+09,9E+09,9E+09,9E+09,9E+09,9E+09]], vmax, z0, tWeldGun;
		ArcLStart [[860.21,550.17,-4.16],[0.152159,0.0392088,0.965632,-0.207039],[0,-2,1,0],[9E+09,9E+09,9E+09,9E+09,9E+09,9E+09]], v20, seam13, weld13\Weave:=weave1, fine, tWeldGun;
		ArcLEnd [[895.96,549.20,-3.18],[0.152141,0.039174,0.965634,-0.207051],[0,-2,1,0],[9E+09,9E+09,9E+09,9E+09,9E+09,9E+09]], v20, seam13, weld13\Weave:=weave1, fine, tWeldGun;
		MoveL [[895.37,549.34,9.83],[0.15211,0.0392827,0.965635,-0.207047],[0,-2,1,0],[9E+09,9E+09,9E+09,9E+09,9E+09,9E+09]], vmax, z0, tWeldGun;
		MoveL [[1175.32,546.94,11.83],[0.1496,0.0478929,0.95235,-0.261449],[0,-2,1,0],[9E+09,9E+09,9E+09,9E+09,9E+09,9E+09]], vmax, z0, tWeldGun;
		ArcLStart [[1177.31,546.94,-3.16],[0.149595,0.0478934,0.95235,-0.261454],[0,-2,1,0],[9E+09,9E+09,9E+09,9E+09,9E+09,9E+09]], v20, seam13, weld13\Weave:=weave1, fine, tWeldGun;
		ArcLEnd [[1209.31,546.95,-3.16],[0.149595,0.0478909,0.95235,-0.261454],[0,-2,1,0],[9E+09,9E+09,9E+09,9E+09,9E+09,9E+09]], v20, seam13, weld13\Weave:=weave1, fine, tWeldGun;
		MoveL [[1183.76,537.75,320.86],[0.152128,0.0394118,0.965637,-0.207003],[0,-2,1,0],[9E+09,9E+09,9E+09,9E+09,9E+09,9E+09]], vmax, z0, tWeldGun;
		MoveJ [[759.22,820.77,477.02],[0.128857,0.0495447,0.958803,-0.24827],[0,-1,1,0],[9E+09,9E+09,9E+09,9E+09,9E+09,9E+09]], vmax, z0, tWeldGun;
		MoveJ [[-401.88,982.38,420.80],[0.377905,-0.177501,-0.908663,-0.00353082],[1,0,1,0],[9E+09,9E+09,9E+09,9E+09,9E+09,9E+09]], vmax, z0, tWeldGun;
		MoveL [[-401.87,982.37,-5.96],[0.377901,-0.177501,-0.908665,-0.00352363],[1,0,1,0],[9E+09,9E+09,9E+09,9E+09,9E+09,9E+09]], v1000, z0, tWeldGun;
		ArcLStart [[-407.18,982.54,-5.95],[0.377941,-0.177364,-0.908675,-0.00361829],[1,0,1,0],[9E+09,9E+09,9E+09,9E+09,9E+09,9E+09]], v10, seam13, weld13\Weave:=weave1, fine, tWeldGun;
		ArcL [[-407.21,961.97,-7.34],[0.377917,-0.177516,-0.908656,-0.00352015],[1,0,1,0],[9E+09,9E+09,9E+09,9E+09,9E+09,9E+09]], v10, seam13, weld13\Weave:=weave1, z10, tWeldGun;
		ArcLEnd [[-429.48,955.83,-6.96],[0.274941,-0.581479,-0.743555,-0.1828],[1,0,2,0],[9E+09,9E+09,9E+09,9E+09,9E+09,9E+09]], v10, seam13, weld13\Weave:=weave1, fine, tWeldGun;
		MoveL [[-432.47,945.01,-6.78],[0.274937,-0.581449,-0.743579,-0.182803],[1,0,2,0],[9E+09,9E+09,9E+09,9E+09,9E+09,9E+09]], vmax, z0, tWeldGun;
		MoveL [[-432.39,895.03,94.24],[0.274951,-0.581467,-0.743558,-0.182811],[1,0,2,0],[9E+09,9E+09,9E+09,9E+09,9E+09,9E+09]], vmax, z0, tWeldGun;
		MoveL [[-1101.20,895.02,94.24],[0.274939,-0.581469,-0.743563,-0.182805],[1,0,2,0],[9E+09,9E+09,9E+09,9E+09,9E+09,9E+09]], vmax, z0, tWeldGun;
		MoveL [[-1101.21,942.37,-3.25],[0.274946,-0.581512,-0.743526,-0.182807],[1,0,2,0],[9E+09,9E+09,9E+09,9E+09,9E+09,9E+09]], v1000, z0, tWeldGun;
		ArcLStart [[-1099.81,952.01,-6.02],[0.23841,-0.593999,-0.734594,-0.225162],[1,0,2,0],[9E+09,9E+09,9E+09,9E+09,9E+09,9E+09]], v10, seam13, weld13\Weave:=weave1, fine, tWeldGun;
		ArcL [[-1121.08,951.80,-5.63],[0.238289,-0.634044,-0.696044,-0.238181],[1,0,2,0],[9E+09,9E+09,9E+09,9E+09,9E+09,9E+09]], v10, seam13, weld13\Weave:=weave1, z10, tWeldGun;
		ArcLEnd [[-1129.28,975.89,-6.00],[0.0369776,0.92297,0.0835389,0.373873],[1,0,3,0],[9E+09,9E+09,9E+09,9E+09,9E+09,9E+09]], v10, seam13, weld13\Weave:=weave1, fine, tWeldGun;
		MoveL [[-1142.99,977.01,6.44],[0.0501214,0.923455,0.0523108,0.376805],[1,0,3,0],[9E+09,9E+09,9E+09,9E+09,9E+09,9E+09]], vmax, z0, tWeldGun;
		MoveJ [[-1142.58,979.31,303.50],[0.0444513,0.923112,0.0666342,0.376096],[1,0,-1,0],[9E+09,9E+09,9E+09,9E+09,9E+09,9E+09]], vmax, z20, tWeldGun;
		MoveL [[-1192.76,1156.53,-4.42],[0.044443,0.923122,0.0666432,0.376072],[1,0,-1,0],[9E+09,9E+09,9E+09,9E+09,9E+09,9E+09]], v1000, z0, tWeldGun;
		ArcLStart [[-1192.23,1155.72,-3.63],[0.0444473,0.923132,0.0666323,0.376048],[1,0,-1,0],[9E+09,9E+09,9E+09,9E+09,9E+09,9E+09]], v10, seam13, weld13\Weave:=weave1, fine, tWeldGun;
		ArcL [[-1191.71,1175.69,-5.33],[0.0444379,0.923126,0.0666324,0.376065],[1,0,-1,0],[9E+09,9E+09,9E+09,9E+09,9E+09,9E+09]], v10, seam13, weld13\Weave:=weave1, z10, tWeldGun;
		ArcLEnd [[-1165.81,1187.00,-4.44],[0.28905,0.665936,-0.622204,0.292989],[1,0,0,0],[9E+09,9E+09,9E+09,9E+09,9E+09,9E+09]], v10, seam13, weld13\Weave:=weave1, fine, tWeldGun;
		MoveL [[-1165.81,1197.81,-4.44],[0.289046,0.665942,-0.622199,0.292988],[1,0,0,0],[9E+09,9E+09,9E+09,9E+09,9E+09,9E+09]], vmax, z0, tWeldGun;
		MoveL [[-1167.37,1197.80,267.48],[0.269054,0.631082,-0.684208,0.247398],[1,-1,0,0],[9E+09,9E+09,9E+09,9E+09,9E+09,9E+09]], vmax, z0, tWeldGun;
		MoveJ [[-491.85,1197.38,267.48],[0.269045,0.631086,-0.684208,0.247399],[1,-1,0,0],[9E+09,9E+09,9E+09,9E+09,9E+09,9E+09]], vmax, z0, tWeldGun;
		MoveL [[-495.49,1197.07,-6.30],[0.260132,0.661057,-0.654909,0.257739],[1,-1,0,0],[9E+09,9E+09,9E+09,9E+09,9E+09,9E+09]], v1000, z0, tWeldGun;
		ArcLStart [[-495.49,1192.07,-6.30],[0.260133,0.661061,-0.654906,0.257736],[1,-1,0,0],[9E+09,9E+09,9E+09,9E+09,9E+09,9E+09]], v10, seam13, weld13\Weave:=weave1, fine, tWeldGun;
		ArcL [[-474.53,1190.57,-6.48],[0.263861,0.655019,-0.660957,0.253897],[1,-1,0,0],[9E+09,9E+09,9E+09,9E+09,9E+09,9E+09]], v10, seam13, weld13\Weave:=weave1, z10, tWeldGun;
		ArcLEnd [[-467.21,1164.88,-8.10],[0.384925,0.00804232,-0.922637,-0.0225898],[1,-1,1,0],[9E+09,9E+09,9E+09,9E+09,9E+09,9E+09]], v10, seam13, weld13\Weave:=weave1, fine, tWeldGun;
		MoveL [[-460.21,1166.10,-6.29],[0.384934,0.00803439,-0.922633,-0.0226006],[1,-1,1,0],[9E+09,9E+09,9E+09,9E+09,9E+09,9E+09]], vmax, z5, tWeldGun;
		MoveL [[-460.61,1166.12,771.55],[0.384916,0.00803537,-0.92264,-0.0226078],[1,-1,1,0],[9E+09,9E+09,9E+09,9E+09,9E+09,9E+09]], vmax, z5, tWeldGun;
		MoveJ pSafeS1, vmax, fine, tWeldGun;
	ENDPROC

	PROC rRUNSIDE1A100()
		MoveJ [[895.91,925.45,959.23],[0.222593,0.0151737,0.948305,-0.225698],[0,-1,0,0],[9E+09,9E+09,9E+09,9E+09,9E+09,9E+09]], vmax, z50, tWeldGun;
		MoveJ [[1169.38,1081.61,325.39],[0.296115,-0.947077,-0.052822,0.112127],[0,-2,0,1],[9E+09,9E+09,9E+09,9E+09,9E+09,9E+09]], vmax, z50, tWeldGun;
		MoveL [[1189.00,1080.17,4.63],[0.333707,-0.921868,0.118398,-0.157423],[0,-2,-1,1],[9E+09,9E+09,9E+09,9E+09,9E+09,9E+09]], v1000, z50, tWeldGun;
		ArcLStart [[1189.77,1081.15,-9.31],[0.333708,-0.921874,0.1184,-0.157385],[0,-2,-1,1],[9E+09,9E+09,9E+09,9E+09,9E+09,9E+09]], v10, seam13, weld13\Weave:=weave1, fine, tWeldGun;
		ArcLEnd [[1155.36,1080.96,-9.32],[0.333709,-0.921872,0.118413,-0.157384],[0,-2,-1,1],[9E+09,9E+09,9E+09,9E+09,9E+09,9E+09]], v10, seam13, weld13\Weave:=weave1, fine, tWeldGun;
		MoveL [[1157.55,1079.96,5.67],[0.333709,-0.921874,0.118398,-0.157383],[0,-2,-1,1],[9E+09,9E+09,9E+09,9E+09,9E+09,9E+09]], vmax, z5, tWeldGun;
		MoveL [[867.14,1075.23,8.88],[0.379709,-0.916742,-0.0425212,0.116612],[0,-2,-1,1],[9E+09,9E+09,9E+09,9E+09,9E+09,9E+09]], vmax, z5, tWeldGun;
		ArcLStart [[867.14,1076.23,-4.29],[0.379693,-0.916748,-0.0425036,0.116619],[0,-2,-1,1],[9E+09,9E+09,9E+09,9E+09,9E+09,9E+09]], v10, seam13, weld13\Weave:=weave1, fine, tWeldGun;
		ArcLEnd [[834.55,1076.01,-3.89],[0.379693,-0.916748,-0.0425149,0.116621],[0,-2,-1,1],[9E+09,9E+09,9E+09,9E+09,9E+09,9E+09]], v10, seam13, weld13\Weave:=weave1, fine, tWeldGun;
		MoveL [[834.56,1075.21,12.06],[0.379682,-0.916754,-0.0425092,0.116603],[0,-2,-1,1],[9E+09,9E+09,9E+09,9E+09,9E+09,9E+09]], vmax, z5, tWeldGun;
		MoveL [[175.01,1076.71,9.09],[0.37968,-0.916766,-0.0425174,0.116513],[0,-2,-1,1],[9E+09,9E+09,9E+09,9E+09,9E+09,9E+09]], vmax, z5, tWeldGun;
		ArcLStart [[175.21,1078.51,-3.72],[0.379675,-0.916769,-0.0425118,0.116508],[0,-2,-1,1],[9E+09,9E+09,9E+09,9E+09,9E+09,9E+09]], v10, seam13, weld13\Weave:=weave1, fine, tWeldGun;
		ArcLEnd [[141.33,1079.10,-3.72],[0.379676,-0.91677,-0.0425113,0.116506],[0,-2,-1,1],[9E+09,9E+09,9E+09,9E+09,9E+09,9E+09]], v10, seam13, weld13\Weave:=weave1, fine, tWeldGun;
		MoveL [[140.80,1076.70,8.09],[0.37968,-0.916765,-0.0425275,0.116517],[0,-2,-1,1],[9E+09,9E+09,9E+09,9E+09,9E+09,9E+09]], vmax, z5, tWeldGun;
		MoveL [[-142.04,1078.78,10.05],[0.379684,-0.916763,-0.0426251,0.116487],[0,-2,-1,1],[9E+09,9E+09,9E+09,9E+09,9E+09,9E+09]], vmax, z5, tWeldGun;
		ArcLStart [[-142.04,1079.38,-3.35],[0.379682,-0.916764,-0.0426296,0.116487],[0,-2,-1,1],[9E+09,9E+09,9E+09,9E+09,9E+09,9E+09]], v10, seam13, weld13\Weave:=weave1, fine, tWeldGun;
		ArcLEnd [[-176.44,1079.18,-3.34],[0.379684,-0.916763,-0.0426122,0.116489],[0,-1,-1,1],[9E+09,9E+09,9E+09,9E+09,9E+09,9E+09]], v10, seam13, weld13\Weave:=weave1, fine, tWeldGun;
		SingArea\Wrist;
		MoveL [[-200.44,1085.42,415.26],[0.379667,-0.916774,-0.042596,0.116465],[0,-2,-1,1],[9E+09,9E+09,9E+09,9E+09,9E+09,9E+09]], vmax, z5, tWeldGun;
		MoveJ [[-173.57,559.75,42.74],[0.145109,0.845875,-0.418866,0.296634],[1,0,-1,0],[9E+09,9E+09,9E+09,9E+09,9E+09,9E+09]], vmax, z5, tWeldGun;
		MoveL [[-169.05,562.52,5.19],[0.145175,0.84585,-0.418945,0.296559],[1,0,-1,0],[9E+09,9E+09,9E+09,9E+09,9E+09,9E+09]], vmax, z5, tWeldGun;
		ArcLStart [[-169.04,560.92,-10.02],[0.145172,0.845851,-0.41894,0.296566],[1,0,-1,0],[9E+09,9E+09,9E+09,9E+09,9E+09,9E+09]], v10, seam13, weld13\Weave:=weave1, fine, tWeldGun;
		ArcLEnd [[-135.88,561.25,-8.17],[0.145137,0.845866,-0.418918,0.296573],[1,0,-1,0],[9E+09,9E+09,9E+09,9E+09,9E+09,9E+09]], v10, seam13, weld13\Weave:=weave1, fine, tWeldGun;
		MoveL [[-136.07,560.62,5.61],[0.145144,0.845861,-0.418915,0.296587],[1,0,-1,0],[9E+09,9E+09,9E+09,9E+09,9E+09,9E+09]], vmax, z5, tWeldGun;
		MoveL [[150.30,559.29,2.38],[0.145275,0.845824,-0.41897,0.296549],[0,0,-1,0],[9E+09,9E+09,9E+09,9E+09,9E+09,9E+09]], vmax, z5, tWeldGun;
		ArcLStart [[149.09,560.10,-11.01],[0.145292,0.845814,-0.419001,0.296528],[0,0,-1,0],[9E+09,9E+09,9E+09,9E+09,9E+09,9E+09]], v10, seam13, weld13\Weave:=weave1, fine, tWeldGun;
		ArcLEnd [[180.89,559.95,-10.61],[0.145283,0.845819,-0.418984,0.29654],[0,0,-1,0],[9E+09,9E+09,9E+09,9E+09,9E+09,9E+09]], v10, seam13, weld13\Weave:=weave1, fine, tWeldGun;
		MoveL [[182.55,560.08,7.18],[0.145153,0.845838,-0.418979,0.296555],[0,0,-1,0],[9E+09,9E+09,9E+09,9E+09,9E+09,9E+09]], vmax, z5, tWeldGun;
		MoveL [[840.66,556.48,0.81],[0.145089,0.845777,-0.419076,0.296625],[0,0,-2,0],[9E+09,9E+09,9E+09,9E+09,9E+09,9E+09]], vmax, z5, tWeldGun;
		ArcLStart [[840.24,557.46,-11.97],[0.145114,0.84576,-0.419121,0.296598],[0,0,-2,0],[9E+09,9E+09,9E+09,9E+09,9E+09,9E+09]], v10, seam13, weld13\Weave:=weave1, fine, tWeldGun;
		ArcLEnd [[872.64,557.26,-12.36],[0.145124,0.845757,-0.419128,0.296591],[0,0,-2,0],[9E+09,9E+09,9E+09,9E+09,9E+09,9E+09]], v10, seam13, weld13\Weave:=weave1, fine, tWeldGun;
		MoveL [[873.71,556.66,3.18],[0.145059,0.845775,-0.419071,0.296652],[0,0,-2,0],[9E+09,9E+09,9E+09,9E+09,9E+09,9E+09]], vmax, z5, tWeldGun;
		MoveL [[1157.38,557.31,-2.39],[0.145019,0.845787,-0.419038,0.296683],[0,0,-2,0],[9E+09,9E+09,9E+09,9E+09,9E+09,9E+09]], vmax, z5, tWeldGun;
		ArcLStart [[1159.14,556.83,-14.78],[0.145041,0.845777,-0.419072,0.296654],[0,0,-2,0],[9E+09,9E+09,9E+09,9E+09,9E+09,9E+09]], v10, seam13, weld13\Weave:=weave1, fine, tWeldGun;
		ArcLEnd [[1191.14,556.43,-14.78],[0.145042,0.845778,-0.41907,0.296654],[0,0,-2,0],[9E+09,9E+09,9E+09,9E+09,9E+09,9E+09]], v10, seam13, weld13\Weave:=weave1, fine, tWeldGun;
		MoveL [[1189.43,560.09,663.81],[0.145007,0.845796,-0.418995,0.296726],[0,0,-2,0],[9E+09,9E+09,9E+09,9E+09,9E+09,9E+09]], vmax, z5, tWeldGun;
		MoveJ [[-229.23,1115.81,554.88],[0.237488,0.691166,-0.628837,0.265431],[1,-1,-4,0],[9E+09,9E+09,9E+09,9E+09,9E+09,9E+09]], vmax, z5, tWeldGun;
		MoveL [[-412.06,717.19,27.71],[0.270403,0.66951,-0.638814,0.265624],[1,0,-4,0],[9E+09,9E+09,9E+09,9E+09,9E+09,9E+09]], vmax, z5, tWeldGun;
		MoveL [[-412.07,716.59,-4.48],[0.270405,0.66951,-0.638815,0.26562],[1,0,-4,0],[9E+09,9E+09,9E+09,9E+09,9E+09,9E+09]], vmax, z5, tWeldGun;
		ArcLStart [[-410.88,712.08,-6.38],[0.270414,0.669517,-0.638809,0.265608],[1,0,-4,0],[9E+09,9E+09,9E+09,9E+09,9E+09,9E+09]], v5, seam13, weld13\Weave:=weave1, fine, tWeldGun;
		ArcLEnd [[-432.89,712.28,-6.37],[0.270423,0.669509,-0.638813,0.265609],[1,0,-4,0],[9E+09,9E+09,9E+09,9E+09,9E+09,9E+09]], v5, seam13, weld13\Weave:=weave1, fine, tWeldGun;
		MoveL [[-435.86,714.19,97.74],[0.270409,0.669504,-0.638821,0.265617],[1,0,-4,0],[9E+09,9E+09,9E+09,9E+09,9E+09,9E+09]], vmax, z5, tWeldGun;
		MoveL [[-1100.50,721.09,94.11],[0.270393,0.669535,-0.638788,0.265635],[1,-1,-4,0],[9E+09,9E+09,9E+09,9E+09,9E+09,9E+09]], vmax, z5, tWeldGun;
		MoveL [[-1101.50,713.37,5.61],[0.270374,0.669541,-0.638766,0.265689],[1,-1,-4,0],[9E+09,9E+09,9E+09,9E+09,9E+09,9E+09]], vmax, z5, tWeldGun;
		ArcLStart [[-1101.59,711.00,-6.35],[0.270404,0.669545,-0.638776,0.265626],[1,-1,-4,0],[9E+09,9E+09,9E+09,9E+09,9E+09,9E+09]], v5, seam13, weld13\Weave:=weave1, fine, tWeldGun;
		ArcLEnd [[-1124.75,711.02,-5.59],[0.270396,0.669535,-0.638784,0.265639],[1,-1,-4,0],[9E+09,9E+09,9E+09,9E+09,9E+09,9E+09]], v5, seam13, weld13\Weave:=weave1, fine, tWeldGun;
		MoveL [[-1124.97,712.38,115.49],[0.270384,0.669531,-0.638781,0.26567],[1,-1,-4,0],[9E+09,9E+09,9E+09,9E+09,9E+09,9E+09]], vmax, z5, tWeldGun;
		MoveJ [[-1119.62,941.62,98.59],[0.263153,-0.665669,-0.65042,-0.254146],[1,0,-2,0],[9E+09,9E+09,9E+09,9E+09,9E+09,9E+09]], vmax, z5, tWeldGun;
		MoveL [[-1103.53,941.47,2.67],[0.263185,-0.665692,-0.650383,-0.254147],[1,0,-2,0],[9E+09,9E+09,9E+09,9E+09,9E+09,9E+09]], vmax, z5, tWeldGun;
		ArcLStart [[-1101.53,952.26,-6.90],[0.245387,-0.665955,-0.67203,-0.211343],[1,0,-2,0],[9E+09,9E+09,9E+09,9E+09,9E+09,9E+09]], v5, seam13, weld13\Weave:=weave1, fine, tWeldGun;
		ArcL [[-1122.43,951.87,-6.14],[0.230872,-0.677147,-0.664308,-0.216486],[1,0,-2,0],[9E+09,9E+09,9E+09,9E+09,9E+09,9E+09]], v5, seam13, weld13\Weave:=weave1, z10, tWeldGun;
		ArcLEnd [[-1127.07,980.82,-7.97],[0.0249196,0.926224,0.00835047,0.376057],[1,0,-1,0],[9E+09,9E+09,9E+09,9E+09,9E+09,9E+09]], v5, seam13, weld13\Weave:=weave1, fine, tWeldGun;
		MoveL [[-1139.22,985.18,63.09],[0.0198475,0.898734,0.00249906,0.438039],[1,-1,-1,0],[9E+09,9E+09,9E+09,9E+09,9E+09,9E+09]], vmax, z5, tWeldGun;
		MoveL [[-1197.13,1157.81,50.93],[0.0198552,0.898739,0.00250141,0.438027],[1,-1,-1,0],[9E+09,9E+09,9E+09,9E+09,9E+09,9E+09]], vmax, z5, tWeldGun;
		MoveL [[-1193.29,1156.64,0.22],[0.0202314,0.914596,0.00160149,0.40386],[1,0,-1,0],[9E+09,9E+09,9E+09,9E+09,9E+09,9E+09]], vmax, z5, tWeldGun;
		ArcLStart [[-1188.51,1160.66,-6.37],[0.0436828,0.938874,-0.0114567,0.341288],[1,0,-1,0],[9E+09,9E+09,9E+09,9E+09,9E+09,9E+09]], v5, seam13, weld13\Weave:=weave1, fine, tWeldGun;
		ArcL [[-1189.05,1179.87,-6.18],[0.0350835,0.946422,-0.0228383,0.320208],[1,0,-1,0],[9E+09,9E+09,9E+09,9E+09,9E+09,9E+09]], v5, seam13, weld13\Weave:=weave1, z10, tWeldGun;
		ArcLEnd [[-1166.55,1190.82,-6.94],[0.234885,0.673237,-0.666707,0.216986],[1,-1,0,0],[9E+09,9E+09,9E+09,9E+09,9E+09,9E+09]], v5, seam13, weld13\Weave:=weave1, fine, tWeldGun;
		MoveL [[-1164.13,1200.44,93.33],[0.251271,0.657126,-0.66952,0.23831],[1,-1,0,0],[9E+09,9E+09,9E+09,9E+09,9E+09,9E+09]], vmax, z5, tWeldGun;
		MoveJ [[-1176.39,1428.24,109.35],[0.303454,-0.641239,-0.63752,-0.300495],[1,-1,2,0],[9E+09,9E+09,9E+09,9E+09,9E+09,9E+09]], vmax, z5, tWeldGun;
		MoveL [[-1186.25,1425.03,14.49],[0.262685,-0.660467,-0.654292,-0.258229],[1,0,2,0],[9E+09,9E+09,9E+09,9E+09,9E+09,9E+09]], vmax, z5, tWeldGun;
		ArcLStart [[-1186.06,1432.23,-6.69],[0.26269,-0.660477,-0.654283,-0.258223],[1,0,2,0],[9E+09,9E+09,9E+09,9E+09,9E+09,9E+09]], v5, seam13, weld13\Weave:=weave1, fine, tWeldGun;
		ArcLEnd [[-1165.11,1431.89,-8.08],[0.262694,-0.66048,-0.654277,-0.258225],[1,0,2,0],[9E+09,9E+09,9E+09,9E+09,9E+09,9E+09]], v5, seam13, weld13\Weave:=weave1, fine, tWeldGun;
		MoveL [[-1165.10,1427.68,74.68],[0.262682,-0.660472,-0.654289,-0.258226],[1,0,2,0],[9E+09,9E+09,9E+09,9E+09,9E+09,9E+09]], vmax, z5, tWeldGun;
		MoveL [[-495.20,1424.53,122.41],[0.28862,-0.64963,-0.643265,-0.284411],[1,-1,2,0],[9E+09,9E+09,9E+09,9E+09,9E+09,9E+09]], vmax, z5, tWeldGun;
		MoveL [[-494.27,1423.22,-1.34],[0.28862,-0.649626,-0.643269,-0.284412],[1,-1,2,0],[9E+09,9E+09,9E+09,9E+09,9E+09,9E+09]], vmax, z5, tWeldGun;
		ArcLStart [[-494.28,1431.62,-11.72],[0.288618,-0.64967,-0.643228,-0.284408],[1,-1,2,0],[9E+09,9E+09,9E+09,9E+09,9E+09,9E+09]], v5, seam13, weld13\Weave:=weave1, fine, tWeldGun;
		ArcLEnd [[-472.28,1431.43,-11.12],[0.288622,-0.649659,-0.643237,-0.284409],[1,-1,2,0],[9E+09,9E+09,9E+09,9E+09,9E+09,9E+09]], v5, seam13, weld13\Weave:=weave1, fine, tWeldGun;
		MoveL [[-474.36,1424.49,125.44],[0.288603,-0.649678,-0.643228,-0.284403],[1,-1,2,0],[9E+09,9E+09,9E+09,9E+09,9E+09,9E+09]], vmax, z5, tWeldGun;
		MoveJ [[-479.04,1241.31,118.19],[0.268582,0.650118,-0.664304,0.252806],[1,-1,0,0],[9E+09,9E+09,9E+09,9E+09,9E+09,9E+09]], vmax, z5, tWeldGun;
		MoveL [[-495.83,1201.80,-1.90],[0.268594,0.650121,-0.6643,0.252797],[1,-1,0,0],[9E+09,9E+09,9E+09,9E+09,9E+09,9E+09]], vmax, z5, tWeldGun;
		ArcLStart [[-493.23,1195.81,-8.08],[0.268589,0.650129,-0.664294,0.252795],[1,-1,0,0],[9E+09,9E+09,9E+09,9E+09,9E+09,9E+09]], v5, seam13, weld13\Weave:=weave1, fine, tWeldGun;
		ArcL [[-475.65,1196.01,-7.47],[0.268596,0.650131,-0.664293,0.252787],[1,-1,0,0],[9E+09,9E+09,9E+09,9E+09,9E+09,9E+09]], v5, seam13, weld13\Weave:=weave1, z10, tWeldGun;
		ArcLEnd [[-468.30,1167.75,-9.67],[0.390504,0.0535497,-0.919043,-0.000178963],[1,-1,1,0],[9E+09,9E+09,9E+09,9E+09,9E+09,9E+09]], v5, seam13, weld13\Weave:=weave1, fine, tWeldGun;
		MoveL [[-435.96,1164.94,59.58],[0.390502,0.0535497,-0.919044,-0.000186584],[1,-1,1,0],[9E+09,9E+09,9E+09,9E+09,9E+09,9E+09]], vmax, z5, tWeldGun;
		MoveL [[-398.53,986.99,7.96],[0.390518,0.0535228,-0.919039,-0.00018247],[1,-1,1,0],[9E+09,9E+09,9E+09,9E+09,9E+09,9E+09]], vmax, z5, tWeldGun;
		ArcLStart [[-407.74,987.37,-7.98],[0.390533,0.0535132,-0.919033,-0.000179522],[1,-1,1,0],[9E+09,9E+09,9E+09,9E+09,9E+09,9E+09]], v20, seam13, weld13\Weave:=weave1, fine, tWeldGun;
		ArcL [[-406.86,967.49,-8.33],[0.390542,0.0535142,-0.919029,-0.000188099],[1,-1,1,0],[9E+09,9E+09,9E+09,9E+09,9E+09,9E+09]], v5, seam13, weld13\Weave:=weave1, z10, tWeldGun;
		ArcLEnd [[-428.10,955.08,-6.46],[0.225047,-0.647546,-0.684631,-0.247627],[1,0,2,0],[9E+09,9E+09,9E+09,9E+09,9E+09,9E+09]], v5, seam13, weld13\Weave:=weave1, fine, tWeldGun;
		MoveL [[-432.86,900.19,113.28],[0.289357,-0.647919,-0.645007,-0.283619],[1,-1,2,0],[9E+09,9E+09,9E+09,9E+09,9E+09,9E+09]], vmax, z5, tWeldGun;
		MoveJ [[276.57,1109.67,795.31],[0.28935,-0.647904,-0.645024,-0.283623],[0,0,1,0],[9E+09,9E+09,9E+09,9E+09,9E+09,9E+09]], vmax, z5, tWeldGun;
	ENDPROC
	PROC ProSkid200()
		MoveJ pSafeS1, vmax, fine, tWeldGun;
		MoveL [[-234.96,1621.92,-8.21],[0.194298,-0.276185,-0.910115,-0.24013],[1,-1,1,0],[9E+09,9E+09,9E+09,9E+09,9E+09,9E+09]], vmax, z50, tWeldGun;
		SingArea\Wrist;
		ArcLStart [[-265.19,1628.57,-38.88],[0.243445,-0.67037,-0.655025,-0.249563],[1,0,2,0],[9E+09,9E+09,9E+09,9E+09,9E+09,9E+09]], v40, seam13, weld13, fine, tWeldGun;
		ArcLEnd [[-257.54,1628.57,-38.88],[0.243445,-0.670369,-0.655025,-0.249565],[1,0,2,0],[9E+09,9E+09,9E+09,9E+09,9E+09,9E+09]], v10, seam13, weld13, fine, tWeldGun;
		MoveL [[-258.35,1618.76,-2.87],[0.243441,-0.670362,-0.655032,-0.24957],[1,0,2,0],[9E+09,9E+09,9E+09,9E+09,9E+09,9E+09]], vmax, z20, tWeldGun;
		MoveJ [[-252.87,717.22,166.31],[0.308554,0.634187,-0.646071,0.291883],[1,0,0,0],[9E+09,9E+09,9E+09,9E+09,9E+09,9E+09]], vmax, z20, tWeldGun;
		SingArea\Wrist;
		MoveL [[-273.06,697.08,-39.01],[0.289422,0.639754,-0.670959,0.238254],[1,0,0,0],[9E+09,9E+09,9E+09,9E+09,9E+09,9E+09]], vmax, z20, tWeldGun;
		ArcLStart [[-273.06,687.07,-45.02],[0.289425,0.639748,-0.670962,0.238258],[1,0,0,0],[9E+09,9E+09,9E+09,9E+09,9E+09,9E+09]], v10, seam13, weld13, fine, tWeldGun;
		ArcLEnd [[-266.46,687.08,-45.02],[0.289425,0.63975,-0.67096,0.238257],[1,0,0,0],[9E+09,9E+09,9E+09,9E+09,9E+09,9E+09]], v10, seam13, weld13, fine, tWeldGun;
		MoveL [[-265.17,697.65,3.08],[0.289425,0.639755,-0.670954,0.238258],[1,0,0,0],[9E+09,9E+09,9E+09,9E+09,9E+09,9E+09]], vmax, z20, tWeldGun;
		MoveJ [[1363.12,672.47,163.81],[0.230647,0.704641,-0.28697,0.606574],[0,-1,-1,0],[9E+09,9E+09,9E+09,9E+09,9E+09,9E+09]], vmax, z20, tWeldGun;
		MoveL [[1363.13,672.48,-59.34],[0.230635,0.704646,-0.28697,0.606573],[0,-1,-1,0],[9E+09,9E+09,9E+09,9E+09,9E+09,9E+09]], vmax, z20, tWeldGun;
		ArcLStart [[1395.10,665.67,-59.36],[0.230647,0.704646,-0.286968,0.606569],[0,-1,-1,0],[9E+09,9E+09,9E+09,9E+09,9E+09,9E+09]], v10, seam13, weld13, fine, tWeldGun;
		ArcLEnd [[1393.21,666.82,-105.76],[0.230653,0.704647,-0.286991,0.606554],[0,-1,-1,0],[9E+09,9E+09,9E+09,9E+09,9E+09,9E+09]], v10, seam13, weld13, fine, tWeldGun;
		MoveL [[1360.51,678.95,-105.76],[0.230657,0.704646,-0.286998,0.60655],[0,-1,-1,0],[9E+09,9E+09,9E+09,9E+09,9E+09,9E+09]], vmax, z20, tWeldGun;
		MoveJ [[1360.48,679.11,200.26],[0.227916,0.703475,-0.290109,0.607465],[0,-1,-1,0],[9E+09,9E+09,9E+09,9E+09,9E+09,9E+09]], vmax, z20, tWeldGun;
		MoveJ [[1372.60,1612.03,89.61],[0.238536,-0.688587,-0.26592,-0.631059],[0,-1,-2,0],[9E+09,9E+09,9E+09,9E+09,9E+09,9E+09]], vmax, z20, tWeldGun;
		MoveL [[1372.62,1612.07,-51.09],[0.238534,-0.68856,-0.265944,-0.631079],[0,-1,-2,0],[9E+09,9E+09,9E+09,9E+09,9E+09,9E+09]], vmax, z20, tWeldGun;
		ArcLStart [[1403.05,1622.70,-51.46],[0.238475,-0.688587,-0.265917,-0.631084],[0,-1,-2,0],[9E+09,9E+09,9E+09,9E+09,9E+09,9E+09]], v10, seam13, weld13, fine, tWeldGun;
		ArcLEnd [[1401.72,1623.96,-98.89],[0.23847,-0.688542,-0.266036,-0.631085],[0,-1,-2,0],[9E+09,9E+09,9E+09,9E+09,9E+09,9E+09]], v10, seam13, weld13, fine, tWeldGun;
		MoveL [[1350.78,1600.25,-98.94],[0.23849,-0.68857,-0.265983,-0.631068],[0,-1,-2,0],[9E+09,9E+09,9E+09,9E+09,9E+09,9E+09]], vmax, z20, tWeldGun;
		MoveL [[1286.32,1556.33,142.30],[0.238485,-0.688572,-0.265997,-0.631063],[0,-1,-2,0],[9E+09,9E+09,9E+09,9E+09,9E+09,9E+09]], vmax, z20, tWeldGun;
		MoveJ [[1024.21,1614.84,123.96],[0.621106,-0.285749,-0.670591,-0.287895],[0,0,0,0],[9E+09,9E+09,9E+09,9E+09,9E+09,9E+09]], vmax, z20, tWeldGun;
		MoveL [[1024.31,1614.97,-44.55],[0.621177,-0.285699,-0.670494,-0.288017],[0,0,0,0],[9E+09,9E+09,9E+09,9E+09,9E+09,9E+09]], vmax, z20, tWeldGun;
		ArcLStart [[986.78,1630.52,-48.85],[0.621168,-0.285689,-0.670501,-0.28803],[0,0,0,0],[9E+09,9E+09,9E+09,9E+09,9E+09,9E+09]], v10, seam13, weld13, fine, tWeldGun;
		ArcLEnd [[989.07,1629.80,-94.04],[0.621174,-0.285677,-0.670503,-0.288024],[0,0,0,0],[9E+09,9E+09,9E+09,9E+09,9E+09,9E+09]], v10, seam13, weld13, fine, tWeldGun;
		MoveL [[1031.38,1620.08,-94.06],[0.621173,-0.285694,-0.670496,-0.288025],[0,0,0,0],[9E+09,9E+09,9E+09,9E+09,9E+09,9E+09]], vmax, z20, tWeldGun;
		MoveL [[1050.77,1575.36,86.67],[0.621174,-0.285691,-0.670496,-0.288026],[0,0,0,0],[9E+09,9E+09,9E+09,9E+09,9E+09,9E+09]], vmax, z20, tWeldGun;
		MoveJ [[1013.51,687.74,143.37],[0.59856,0.318284,-0.67023,0.302017],[0,-1,-1,0],[9E+09,9E+09,9E+09,9E+09,9E+09,9E+09]], vmax, z20, tWeldGun;
		MoveL [[1013.45,687.71,-58.15],[0.598615,0.318227,-0.670196,0.302042],[0,-1,-1,0],[9E+09,9E+09,9E+09,9E+09,9E+09,9E+09]], vmax, z20, tWeldGun;
		ArcLStart [[981.75,669.03,-58.14],[0.598616,0.318216,-0.6702,0.302041],[0,-1,-1,0],[9E+09,9E+09,9E+09,9E+09,9E+09,9E+09]], v10, seam13, weld13, fine, tWeldGun;
		ArcLEnd [[981.75,669.03,-102.94],[0.598614,0.318211,-0.670206,0.302041],[0,-1,-1,0],[9E+09,9E+09,9E+09,9E+09,9E+09,9E+09]], v10, seam13, weld13, fine, tWeldGun;
		MoveL [[1021.06,692.65,-100.54],[0.598619,0.318178,-0.670217,0.30204],[0,-1,-1,0],[9E+09,9E+09,9E+09,9E+09,9E+09,9E+09]], vmax, z20, tWeldGun;
		MoveL [[1021.06,692.65,172.93],[0.598621,0.318175,-0.670218,0.302038],[0,-1,-1,0],[9E+09,9E+09,9E+09,9E+09,9E+09,9E+09]], vmax, z20, tWeldGun;
		MoveJ [[962.66,684.38,264.32],[0.236784,0.681997,-0.2918,0.627429],[0,1,1,1],[9E+09,9E+09,9E+09,9E+09,9E+09,9E+09]], vmax, z20, tWeldGun;
		MoveL [[962.64,684.38,-48.75],[0.236792,0.682002,-0.291815,0.627413],[0,1,1,1],[9E+09,9E+09,9E+09,9E+09,9E+09,9E+09]], vmax, z20, tWeldGun;
		ArcLStart [[980.94,668.93,-48.75],[0.236782,0.682005,-0.291808,0.627418],[0,1,1,1],[9E+09,9E+09,9E+09,9E+09,9E+09,9E+09]], v10, seam13, weld13, fine, tWeldGun;
		ArcLEnd [[980.92,669.75,-104.66],[0.236799,0.682008,-0.291831,0.627396],[0,1,1,1],[9E+09,9E+09,9E+09,9E+09,9E+09,9E+09]], v10, seam13, weld13, fine, tWeldGun;
		MoveL [[948.38,696.75,-105.45],[0.234731,0.68317,-0.291592,0.62702],[0,1,1,1],[9E+09,9E+09,9E+09,9E+09,9E+09,9E+09]], vmax, z20, tWeldGun;
		MoveL [[948.40,696.76,143.62],[0.234722,0.683169,-0.291572,0.627035],[0,1,1,1],[9E+09,9E+09,9E+09,9E+09,9E+09,9E+09]], vmax, z20, tWeldGun;
		MoveJ [[975.43,1612.68,308.57],[0.225877,-0.689512,-0.28382,-0.626896],[0,1,0,1],[9E+09,9E+09,9E+09,9E+09,9E+09,9E+09]], vmax, z20, tWeldGun;
		MoveL [[975.55,1612.35,-40.05],[0.22557,-0.689612,-0.283854,-0.626882],[0,0,1,1],[9E+09,9E+09,9E+09,9E+09,9E+09,9E+09]], vmax, z20, tWeldGun;
		ArcLStart [[989.75,1627.18,-40.10],[0.225683,-0.689679,-0.283801,-0.626791],[0,1,1,1],[9E+09,9E+09,9E+09,9E+09,9E+09,9E+09]], v10, seam13, weld13, fine, tWeldGun;
		ArcLEnd [[988.02,1626.51,-103.36],[0.218861,-0.704472,-0.289009,-0.610159],[0,1,1,1],[9E+09,9E+09,9E+09,9E+09,9E+09,9E+09]], v10, seam13, weld13, fine, tWeldGun;
		MoveL [[969.19,1616.42,-103.36],[0.21886,-0.704489,-0.288978,-0.610154],[0,1,1,1],[9E+09,9E+09,9E+09,9E+09,9E+09,9E+09]], vmax, z20, tWeldGun;
		MoveL [[972.04,1615.87,168.33],[0.225681,-0.689708,-0.283758,-0.62678],[0,1,0,1],[9E+09,9E+09,9E+09,9E+09,9E+09,9E+09]], vmax, z20, tWeldGun;
		MoveJ [[748.32,1594.78,-28.74],[0.231269,-0.620927,-0.702805,-0.258902],[0,1,-1,1],[9E+09,9E+09,9E+09,9E+09,9E+09,9E+09]], vmax, z20, tWeldGun;
		MoveL [[748.32,1618.27,-62.58],[0.231267,-0.620927,-0.702807,-0.258898],[0,1,-1,1],[9E+09,9E+09,9E+09,9E+09,9E+09,9E+09]], vmax, z20, tWeldGun;
		ArcLStart [[748.35,1622.75,-67.83],[0.23126,-0.620915,-0.702812,-0.25892],[0,1,-1,1],[9E+09,9E+09,9E+09,9E+09,9E+09,9E+09]], v10, seam13, weld13, fine, tWeldGun;
		ArcLEnd [[720.93,1622.75,-67.82],[0.231262,-0.620925,-0.702803,-0.258918],[0,1,-1,1],[9E+09,9E+09,9E+09,9E+09,9E+09,9E+09]], v10, seam13, weld13, fine, tWeldGun;
		MoveL [[683.13,1622.94,-67.84],[0.231262,-0.620938,-0.702794,-0.258913],[0,1,-1,1],[9E+09,9E+09,9E+09,9E+09,9E+09,9E+09]], vmax, z20, tWeldGun;
		ArcLStart [[681.00,1622.93,-67.87],[0.231258,-0.62095,-0.702784,-0.258913],[0,1,-1,1],[9E+09,9E+09,9E+09,9E+09,9E+09,9E+09]], v10, seam13, weld13, fine, tWeldGun;
		ArcLEnd [[654.73,1623.14,-67.84],[0.231266,-0.620945,-0.702787,-0.258912],[0,1,-1,1],[9E+09,9E+09,9E+09,9E+09,9E+09,9E+09]], v10, seam13, weld13, fine, tWeldGun;
		MoveL [[654.72,1619.33,-13.30],[0.231269,-0.620959,-0.702776,-0.258903],[0,1,-1,1],[9E+09,9E+09,9E+09,9E+09,9E+09,9E+09]], vmax, z20, tWeldGun;
		MoveJ [[37.05,1622.28,-7.90],[0.231269,-0.620971,-0.702762,-0.258912],[1,1,-1,1],[9E+09,9E+09,9E+09,9E+09,9E+09,9E+09]], vmax, z20, tWeldGun;
		MoveL [[37.06,1622.28,-65.61],[0.231267,-0.620964,-0.702769,-0.258912],[1,1,-1,1],[9E+09,9E+09,9E+09,9E+09,9E+09,9E+09]], vmax, z20, tWeldGun;
		ArcLStart [[37.05,1628.08,-65.61],[0.231271,-0.620973,-0.702759,-0.258914],[1,1,-1,1],[9E+09,9E+09,9E+09,9E+09,9E+09,9E+09]], v10, seam13, weld13, fine, tWeldGun;
		ArcLEnd [[7.65,1628.68,-65.60],[0.231271,-0.620979,-0.702755,-0.258912],[1,1,-1,1],[9E+09,9E+09,9E+09,9E+09,9E+09,9E+09]], v10, seam13, weld13, fine, tWeldGun;
		MoveL [[-27.35,1629.08,-65.60],[0.231271,-0.620982,-0.702752,-0.258911],[1,1,0,1],[9E+09,9E+09,9E+09,9E+09,9E+09,9E+09]], vmax, z20, tWeldGun;
		ArcLStart [[-31.75,1629.08,-65.60],[0.231272,-0.620988,-0.702747,-0.258912],[1,1,0,1],[9E+09,9E+09,9E+09,9E+09,9E+09,9E+09]], v10, seam13, weld13, fine, tWeldGun;
		ArcLEnd [[-60.36,1629.07,-65.63],[0.231269,-0.621009,-0.70273,-0.258909],[1,1,0,1],[9E+09,9E+09,9E+09,9E+09,9E+09,9E+09]], v10, seam13, weld13, fine, tWeldGun;
		MoveL [[-63.19,1451.21,44.92],[0.231265,-0.62101,-0.702733,-0.258902],[1,1,0,1],[9E+09,9E+09,9E+09,9E+09,9E+09,9E+09]], vmax, z20, tWeldGun;
		SingArea\Wrist;
		MoveJ [[-220.42,1456.39,142.20],[0.365991,-0.606888,-0.673424,-0.210328],[1,0,1,0],[9E+09,9E+09,9E+09,9E+09,9E+09,9E+09]], vmax, z20, tWeldGun;
		MoveL [[-219.91,1623.63,-54.86],[0.365978,-0.606856,-0.673457,-0.210339],[1,0,1,0],[9E+09,9E+09,9E+09,9E+09,9E+09,9E+09]], vmax, z20, tWeldGun;
		ArcLStart [[-219.83,1630.03,-63.47],[0.36598,-0.606851,-0.67346,-0.21034],[1,0,1,0],[9E+09,9E+09,9E+09,9E+09,9E+09,9E+09]], v10, seam13, weld13, fine, tWeldGun;
		ArcLEnd [[-233.82,1630.03,-62.87],[0.365977,-0.606844,-0.673467,-0.210341],[1,0,1,0],[9E+09,9E+09,9E+09,9E+09,9E+09,9E+09]], v10, seam13, weld13, fine, tWeldGun;
		MoveL [[-229.83,1622.04,44.03],[0.365923,-0.606933,-0.673436,-0.21028],[1,0,1,0],[9E+09,9E+09,9E+09,9E+09,9E+09,9E+09]], vmax, z20, tWeldGun;
		MoveJ [[-238.42,695.07,107.36],[0.416175,0.412803,-0.798145,0.139133],[1,0,0,0],[9E+09,9E+09,9E+09,9E+09,9E+09,9E+09]], vmax, z20, tWeldGun;
		MoveL [[-238.43,695.09,-59.53],[0.416176,0.412786,-0.798155,0.139122],[1,0,0,0],[9E+09,9E+09,9E+09,9E+09,9E+09,9E+09]], vmax, z20, tWeldGun;
		ArcLStart [[-240.41,687.67,-69.36],[0.416165,0.412798,-0.798152,0.139137],[1,0,0,0],[9E+09,9E+09,9E+09,9E+09,9E+09,9E+09]], v10, seam13, weld13, fine, tWeldGun;
		ArcLEnd [[-225.81,687.67,-69.75],[0.416158,0.41281,-0.798148,0.139143],[1,0,0,0],[9E+09,9E+09,9E+09,9E+09,9E+09,9E+09]], v10, seam13, weld13, fine, tWeldGun;
		MoveL [[-226.30,704.95,-17.45],[0.416163,0.412818,-0.79814,0.139151],[1,0,0,0],[9E+09,9E+09,9E+09,9E+09,9E+09,9E+09]], vmax, z20, tWeldGun;
		MoveJ [[-68.54,708.92,-17.46],[0.33715,0.641758,-0.612556,0.315044],[1,0,-1,0],[9E+09,9E+09,9E+09,9E+09,9E+09,9E+09]], vmax, z20, tWeldGun;
		MoveL [[-69.37,694.59,-61.82],[0.293998,0.661849,-0.635411,0.267907],[1,0,-1,0],[9E+09,9E+09,9E+09,9E+09,9E+09,9E+09]], vmax, z20, tWeldGun;
		ArcLStart [[-69.36,687.96,-70.31],[0.294028,0.661818,-0.635424,0.26792],[1,0,-1,0],[9E+09,9E+09,9E+09,9E+09,9E+09,9E+09]], v10, seam13, weld13, fine, tWeldGun;
		ArcLEnd [[-41.96,687.95,-70.52],[0.29404,0.66181,-0.635427,0.267921],[1,0,-1,0],[9E+09,9E+09,9E+09,9E+09,9E+09,9E+09]], v10, seam13, weld13, fine, tWeldGun;
		MoveL [[-6.97,687.95,-70.51],[0.294043,0.661806,-0.635431,0.267916],[0,0,-1,0],[9E+09,9E+09,9E+09,9E+09,9E+09,9E+09]], vmax, z20, tWeldGun;
		ArcLStart [[-6.96,687.54,-70.52],[0.294045,0.661806,-0.635429,0.267919],[0,0,-1,0],[9E+09,9E+09,9E+09,9E+09,9E+09,9E+09]], v10, seam13, weld13, fine, tWeldGun;
		ArcLEnd [[21.80,686.99,-70.51],[0.294054,0.661794,-0.635442,0.267908],[0,0,-1,0],[9E+09,9E+09,9E+09,9E+09,9E+09,9E+09]], v10, seam13, weld13, fine, tWeldGun;
		MoveL [[21.80,693.66,-56.32],[0.294011,0.661823,-0.635446,0.267875],[0,0,-1,0],[9E+09,9E+09,9E+09,9E+09,9E+09,9E+09]], vmax, z20, tWeldGun;
		MoveL [[644.60,694.09,-38.11],[0.29406,0.661788,-0.635447,0.267906],[0,0,-1,0],[9E+09,9E+09,9E+09,9E+09,9E+09,9E+09]], vmax, z20, tWeldGun;
		ArcLStart [[644.53,682.78,-73.42],[0.294076,0.661755,-0.635493,0.267859],[0,0,-1,0],[9E+09,9E+09,9E+09,9E+09,9E+09,9E+09]], v40, seam13, weld13, fine, tWeldGun;
		ArcLEnd [[667.66,682.46,-73.44],[0.294106,0.661729,-0.635513,0.267845],[0,0,-1,0],[9E+09,9E+09,9E+09,9E+09,9E+09,9E+09]], v10, seam13, weld13, fine, tWeldGun;
		MoveL [[706.98,682.46,-73.44],[0.294117,0.661731,-0.635507,0.267842],[0,0,-1,0],[9E+09,9E+09,9E+09,9E+09,9E+09,9E+09]], vmax, z20, tWeldGun;
		ArcLStart [[706.98,682.46,-73.44],[0.294117,0.66173,-0.635507,0.267841],[0,0,-1,0],[9E+09,9E+09,9E+09,9E+09,9E+09,9E+09]], v10, seam13, weld13, fine, tWeldGun;
		ArcLEnd [[732.78,682.64,-73.45],[0.294116,0.66175,-0.635481,0.267856],[0,0,-1,0],[9E+09,9E+09,9E+09,9E+09,9E+09,9E+09]], v10, seam13, weld13, fine, tWeldGun;
		MoveL [[743.36,710.11,-13.87],[0.294132,0.661743,-0.635486,0.267845],[0,0,-1,0],[9E+09,9E+09,9E+09,9E+09,9E+09,9E+09]], vmax, z20, tWeldGun;
		MoveJ [[766.73,689.09,12.78],[0.426939,0.266425,-0.809663,0.301972],[0,-1,0,0],[9E+09,9E+09,9E+09,9E+09,9E+09,9E+09]], vmax, z20, tWeldGun;
		MoveL [[766.72,689.01,-73.04],[0.426946,0.266425,-0.809635,0.302037],[0,-1,0,0],[9E+09,9E+09,9E+09,9E+09,9E+09,9E+09]], vmax, z20, tWeldGun;
		ArcLStart [[753.37,674.21,-83.82],[0.426978,0.266403,-0.80963,0.302027],[0,-1,0,0],[9E+09,9E+09,9E+09,9E+09,9E+09,9E+09]], v10, seam13, weld13, fine, tWeldGun;
		ArcLEnd [[753.94,674.20,-111.42],[0.427004,0.266403,-0.809617,0.302024],[0,-1,0,0],[9E+09,9E+09,9E+09,9E+09,9E+09,9E+09]], v10, seam13, weld13, fine, tWeldGun;
		MoveL [[767.24,687.28,-25.85],[0.427002,0.266345,-0.809691,0.301878],[0,-1,0,0],[9E+09,9E+09,9E+09,9E+09,9E+09,9E+09]], vmax, z20, tWeldGun;
		MoveJ [[43.23,696.82,-1.72],[0.42676,0.266354,-0.810055,0.301235],[0,-1,0,0],[9E+09,9E+09,9E+09,9E+09,9E+09,9E+09]], vmax, z20, tWeldGun;
		MoveL [[42.01,683.49,-78.40],[0.427024,0.26632,-0.809694,0.301862],[0,-1,0,0],[9E+09,9E+09,9E+09,9E+09,9E+09,9E+09]], vmax, z20, tWeldGun;
		ArcLStart [[38.82,680.87,-78.40],[0.427033,0.266358,-0.80967,0.301881],[0,-1,0,0],[9E+09,9E+09,9E+09,9E+09,9E+09,9E+09]], v10, seam13, weld13, fine, tWeldGun;
		ArcLEnd [[40.20,680.75,-109.60],[0.427039,0.266382,-0.80967,0.301849],[0,-1,0,0],[9E+09,9E+09,9E+09,9E+09,9E+09,9E+09]], v10, seam13, weld13, fine, tWeldGun;
		MoveL [[56.60,714.15,-11.47],[0.427063,0.266301,-0.809685,0.301848],[0,-1,0,0],[9E+09,9E+09,9E+09,9E+09,9E+09,9E+09]], vmax, z20, tWeldGun;
		MoveJ [[-90.85,716.79,14.15],[0.243321,0.796043,-0.267285,0.485459],[1,-1,-1,0],[9E+09,9E+09,9E+09,9E+09,9E+09,9E+09]], vmax, z20, tWeldGun;
		MoveL [[-92.64,686.16,-78.85],[0.243349,0.796017,-0.267252,0.485505],[1,-1,-1,0],[9E+09,9E+09,9E+09,9E+09,9E+09,9E+09]], vmax, z20, tWeldGun;
		ArcLStart [[-85.54,680.97,-78.85],[0.243338,0.796021,-0.267256,0.485502],[1,-1,-1,0],[9E+09,9E+09,9E+09,9E+09,9E+09,9E+09]], v10, seam13, weld13, fine, tWeldGun;
		ArcLEnd [[-85.54,680.97,-106.06],[0.243338,0.796019,-0.267253,0.485507],[1,-1,-1,0],[9E+09,9E+09,9E+09,9E+09,9E+09,9E+09]], v10, seam13, weld13, fine, tWeldGun;
		MoveL [[-99.62,700.82,-3.32],[0.243332,0.796035,-0.267233,0.485495],[1,-1,-1,0],[9E+09,9E+09,9E+09,9E+09,9E+09,9E+09]], vmax, z20, tWeldGun;
		MoveJ [[622.81,695.86,-3.35],[0.24331,0.796057,-0.26719,0.485493],[0,-1,-1,0],[9E+09,9E+09,9E+09,9E+09,9E+09,9E+09]], vmax, z20, tWeldGun;
		MoveL [[622.81,678.68,-81.59],[0.243312,0.796055,-0.267198,0.485492],[0,-1,-1,0],[9E+09,9E+09,9E+09,9E+09,9E+09,9E+09]], vmax, z20, tWeldGun;
		ArcLStart [[627.79,674.24,-83.40],[0.243343,0.796045,-0.267192,0.485495],[0,-1,-1,0],[9E+09,9E+09,9E+09,9E+09,9E+09,9E+09]], v10, seam13, weld13, fine, tWeldGun;
		ArcLEnd [[626.78,674.63,-109.81],[0.243358,0.796042,-0.267204,0.485485],[0,-1,-1,0],[9E+09,9E+09,9E+09,9E+09,9E+09,9E+09]], v10, seam13, weld13, fine, tWeldGun;
		MoveL [[610.77,692.21,49.90],[0.243321,0.79605,-0.267267,0.485457],[0,-1,-1,0],[9E+09,9E+09,9E+09,9E+09,9E+09,9E+09]], vmax, z20, tWeldGun;
		MoveJ [[622.12,1614.25,159.14],[0.192579,-0.77773,-0.32949,-0.499486],[0,1,0,1],[9E+09,9E+09,9E+09,9E+09,9E+09,9E+09]], vmax, z20, tWeldGun;
		MoveL [[622.15,1614.23,-75.01],[0.192557,-0.777696,-0.329551,-0.499508],[0,1,0,1],[9E+09,9E+09,9E+09,9E+09,9E+09,9E+09]], vmax, z20, tWeldGun;
		ArcLStart [[640.60,1627.79,-79.81],[0.192567,-0.777665,-0.329604,-0.499517],[0,1,0,1],[9E+09,9E+09,9E+09,9E+09,9E+09,9E+09]], v10, seam13, weld13, fine, tWeldGun;
		ArcLEnd [[640.40,1627.75,-105.01],[0.19256,-0.777691,-0.32956,-0.499508],[0,1,0,1],[9E+09,9E+09,9E+09,9E+09,9E+09,9E+09]], v10, seam13, weld13, fine, tWeldGun;
		MoveL [[622.01,1617.53,-16.15],[0.192549,-0.777705,-0.329542,-0.499501],[0,1,0,1],[9E+09,9E+09,9E+09,9E+09,9E+09,9E+09]], vmax, z20, tWeldGun;
		MoveJ [[-74.83,1621.54,-16.16],[0.19255,-0.777728,-0.329501,-0.499493],[1,1,0,1],[9E+09,9E+09,9E+09,9E+09,9E+09,9E+09]], vmax, z20, tWeldGun;
		MoveL [[-74.84,1632.22,-76.43],[0.192546,-0.777738,-0.329487,-0.499489],[1,1,0,1],[9E+09,9E+09,9E+09,9E+09,9E+09,9E+09]], vmax, z20, tWeldGun;
		ArcLStart [[-72.04,1634.00,-74.85],[0.192535,-0.777754,-0.329462,-0.499484],[1,1,0,1],[9E+09,9E+09,9E+09,9E+09,9E+09,9E+09]], v10, seam13, weld13, fine, tWeldGun;
		ArcLEnd [[-72.05,1633.99,-104.27],[0.19253,-0.777762,-0.329453,-0.49948],[1,1,0,1],[9E+09,9E+09,9E+09,9E+09,9E+09,9E+09]], v10, seam13, weld13, fine, tWeldGun;
		MoveL [[-101.85,1558.57,140.36],[0.192608,-0.777808,-0.329372,-0.499431],[1,1,0,1],[9E+09,9E+09,9E+09,9E+09,9E+09,9E+09]], vmax, z20, tWeldGun;
		MoveJ [[102.30,1319.34,116.73],[0.326866,-0.251271,-0.905673,-0.0988914],[0,-1,1,0],[9E+09,9E+09,9E+09,9E+09,9E+09,9E+09]], vmax, z20, tWeldGun;
		MoveL [[56.99,1626.55,-72.67],[0.410474,-0.275782,-0.84185,-0.216205],[0,0,1,0],[9E+09,9E+09,9E+09,9E+09,9E+09,9E+09]], vmax, z20, tWeldGun;
		ArcLStart [[49.28,1632.40,-74.45],[0.41046,-0.275749,-0.841871,-0.216193],[0,0,1,0],[9E+09,9E+09,9E+09,9E+09,9E+09,9E+09]], v10, seam13, weld13, fine, tWeldGun;
		ArcLEnd [[51.27,1632.00,-107.06],[0.410475,-0.275775,-0.841856,-0.216189],[0,0,1,0],[9E+09,9E+09,9E+09,9E+09,9E+09,9E+09]], v10, seam13, weld13, fine, tWeldGun;
		MoveL [[63.32,1618.59,53.83],[0.41045,-0.275792,-0.841833,-0.216304],[0,0,1,0],[9E+09,9E+09,9E+09,9E+09,9E+09,9E+09]], vmax, z20, tWeldGun;
		MoveJ [[774.48,1618.06,-14.91],[0.410442,-0.275748,-0.841846,-0.216328],[0,0,1,0],[9E+09,9E+09,9E+09,9E+09,9E+09,9E+09]], vmax, z20, tWeldGun;
		MoveL [[774.44,1618.01,-79.45],[0.410464,-0.275799,-0.841828,-0.216288],[0,0,0,0],[9E+09,9E+09,9E+09,9E+09,9E+09,9E+09]], vmax, z20, tWeldGun;
		ArcLStart [[760.64,1625.90,-79.46],[0.410464,-0.275804,-0.841826,-0.216291],[0,0,1,0],[9E+09,9E+09,9E+09,9E+09,9E+09,9E+09]], v10, seam13, weld13, fine, tWeldGun;
		ArcLEnd [[761.81,1625.90,-106.65],[0.410464,-0.2758,-0.841828,-0.216289],[0,0,1,0],[9E+09,9E+09,9E+09,9E+09,9E+09,9E+09]], v10, seam13, weld13, fine, tWeldGun;
		MoveL [[783.26,1604.44,251.05],[0.410482,-0.275804,-0.84182,-0.216279],[0,0,1,0],[9E+09,9E+09,9E+09,9E+09,9E+09,9E+09]], vmax, z20, tWeldGun;
		MoveJ pSafeS1, vmax, fine, tWeldGun;
	ENDPROC
	PROC ProSkid50()
		MoveJ [[314.39,1632.04,274.09],[0.410833,-0.611914,-0.675728,-0.0129978],[0,0,-3,0],[9E+09,9E+09,9E+09,9E+09,9E+09,9E+09]], vmax, z50, tWeldGun;
		MoveL [[314.32,1632.00,-25.30],[0.410826,-0.611972,-0.675681,-0.0129369],[0,0,-3,0],[9E+09,9E+09,9E+09,9E+09,9E+09,9E+09]], vmax, z50, tWeldGun;
		ArcLStart [[314.43,1633.11,-39.30],[0.349657,-0.639186,-0.683585,-0.0435139],[0,0,-3,0],[9E+09,9E+09,9E+09,9E+09,9E+09,9E+09]], v10, seam13, weld13, fine, tWeldGun;
		ArcL [[333.87,1632.50,-40.55],[0.349642,-0.639186,-0.683593,-0.0435083],[0,0,-3,0],[9E+09,9E+09,9E+09,9E+09,9E+09,9E+09]], v10, seam13, weld13, z5, tWeldGun;
		ArcL [[341.01,1631.27,-66.17],[0.317739,-0.654055,-0.683899,-0.0594762],[0,0,-3,0],[9E+09,9E+09,9E+09,9E+09,9E+09,9E+09]], v10, seam13, weld13, z5, tWeldGun;
		ArcLEnd [[358.67,1633.28,-65.92],[0.326244,-0.656849,-0.673963,-0.0888224],[0,0,-3,0],[9E+09,9E+09,9E+09,9E+09,9E+09,9E+09]], v10, seam13, weld13, fine, tWeldGun;
		MoveL [[364.49,1617.70,-14.89],[0.410824,-0.611946,-0.675708,-0.012893],[0,0,-3,0],[9E+09,9E+09,9E+09,9E+09,9E+09,9E+09]], vmax, z50, tWeldGun;
		MoveJ [[320.64,789.47,304.99],[0.235374,0.107276,-0.920325,0.293418],[0,-1,-4,0],[9E+09,9E+09,9E+09,9E+09,9E+09,9E+09]], vmax, z50, tWeldGun;
		MoveL [[320.65,680.04,-28.04],[0.235364,0.107285,-0.920324,0.293424],[0,-1,-4,0],[9E+09,9E+09,9E+09,9E+09,9E+09,9E+09]], vmax, z50, tWeldGun;
		ArcLStart [[320.49,676.84,-46.47],[0.235331,0.107401,-0.920274,0.293565],[0,-1,-4,0],[9E+09,9E+09,9E+09,9E+09,9E+09,9E+09]], v10, seam13, weld13, fine, tWeldGun;
		ArcL [[339.64,676.63,-48.64],[0.235361,0.107405,-0.920265,0.293567],[0,-1,-4,0],[9E+09,9E+09,9E+09,9E+09,9E+09,9E+09]], v5, seam13, weld13, z5, tWeldGun;
		ArcL [[342.53,676.66,-71.41],[0.281426,0.0897427,-0.912937,0.281589],[0,-1,-4,0],[9E+09,9E+09,9E+09,9E+09,9E+09,9E+09]], v5, seam13, weld13, z5, tWeldGun;
		ArcLEnd [[360.55,681.94,-73.50],[0.314989,0.316109,-0.866408,0.224044],[0,-1,-4,0],[9E+09,9E+09,9E+09,9E+09,9E+09,9E+09]], v10, seam13, weld13, fine, tWeldGun;
		MoveL [[365.60,682.37,3.04],[0.235347,0.107379,-0.920294,0.293497],[0,-1,-4,0],[9E+09,9E+09,9E+09,9E+09,9E+09,9E+09]], vmax, z50, tWeldGun;
		MoveJ [[836.02,763.37,35.73],[0.0217026,-0.41169,0.816455,-0.40428],[0,-2,-4,0],[9E+09,9E+09,9E+09,9E+09,9E+09,9E+09]], vmax, z50, tWeldGun;
		MoveL [[856.70,689.76,-27.01],[0.0217072,-0.411704,0.816444,-0.404287],[0,-2,-3,0],[9E+09,9E+09,9E+09,9E+09,9E+09,9E+09]], vmax, z50, tWeldGun;
		ArcLStart [[857.91,678.67,-44.98],[0.0203271,-0.414175,0.82252,-0.389238],[0,-2,-3,0],[9E+09,9E+09,9E+09,9E+09,9E+09,9E+09]], v10, seam13, weld13, fine, tWeldGun;
		ArcL [[836.15,679.48,-46.99],[0.0203132,-0.414191,0.822508,-0.389249],[0,-2,-3,0],[9E+09,9E+09,9E+09,9E+09,9E+09,9E+09]], v10, seam13, weld13, z5, tWeldGun;
		ArcL [[831.91,680.96,-69.65],[0.0726329,-0.437948,0.812132,-0.37864],[0,-2,-3,0],[9E+09,9E+09,9E+09,9E+09,9E+09,9E+09]], v10, seam13, weld13, z5, tWeldGun;
		ArcLEnd [[814.71,680.94,-69.65],[0.0726252,-0.437942,0.812135,-0.378643],[0,-2,-3,0],[9E+09,9E+09,9E+09,9E+09,9E+09,9E+09]], v10, seam13, weld13, fine, tWeldGun;
		MoveL [[809.35,725.26,127.04],[0.0216773,-0.411756,0.816405,-0.404315],[0,-2,-4,0],[9E+09,9E+09,9E+09,9E+09,9E+09,9E+09]], vmax, z50, tWeldGun;
		MoveJ [[841.70,1629.86,72.25],[0.220866,-0.864976,-0.348476,-0.285657],[0,0,-2,0],[9E+09,9E+09,9E+09,9E+09,9E+09,9E+09]], vmax, z50, tWeldGun;
		MoveL [[841.69,1629.87,-34.30],[0.220872,-0.864976,-0.348474,-0.285654],[0,0,-2,0],[9E+09,9E+09,9E+09,9E+09,9E+09,9E+09]], vmax, z50, tWeldGun;
		ArcLStart [[848.66,1634.80,-44.07],[0.220862,-0.865006,-0.348435,-0.28562],[0,0,-2,0],[9E+09,9E+09,9E+09,9E+09,9E+09,9E+09]], v20, seam13, weld13, fine, tWeldGun;
		ArcL [[827.08,1634.97,-46.50],[0.220852,-0.865009,-0.348428,-0.285626],[0,0,-2,0],[9E+09,9E+09,9E+09,9E+09,9E+09,9E+09]], v10, seam13, weld13, z1, tWeldGun;
		ArcL [[824.68,1632.91,-69.83],[0.143373,-0.869884,-0.317855,-0.348876],[0,0,-2,0],[9E+09,9E+09,9E+09,9E+09,9E+09,9E+09]], v10, seam13, weld13, z1, tWeldGun;
		ArcLEnd [[803.26,1635.12,-68.75],[0.265625,-0.855119,-0.383795,-0.225647],[0,0,-3,0],[9E+09,9E+09,9E+09,9E+09,9E+09,9E+09]], v10, seam13, weld13, fine, tWeldGun;
		MoveL [[798.38,1604.44,59.29],[0.220844,-0.86502,-0.348413,-0.285617],[0,0,-2,0],[9E+09,9E+09,9E+09,9E+09,9E+09,9E+09]], vmax, z50, tWeldGun;
		MoveJ [[1012.25,1627.55,26.24],[0.148022,-0.852995,-0.305302,-0.396586],[0,-1,-2,0],[9E+09,9E+09,9E+09,9E+09,9E+09,9E+09]], vmax, z50, tWeldGun;
		MoveL [[1012.25,1627.54,-29.96],[0.148013,-0.852994,-0.305304,-0.39659],[0,-1,-2,0],[9E+09,9E+09,9E+09,9E+09,9E+09,9E+09]], vmax, z50, tWeldGun;
		ArcLStart [[1020.33,1635.81,-42.74],[0.234694,-0.797645,-0.305793,-0.463867],[0,0,-2,0],[9E+09,9E+09,9E+09,9E+09,9E+09,9E+09]], v10, seam13, weld13, fine, tWeldGun;
		ArcLEnd [[1020.32,1636.60,-101.76],[0.234691,-0.797653,-0.305783,-0.463861],[0,0,-2,0],[9E+09,9E+09,9E+09,9E+09,9E+09,9E+09]], v10, seam13, weld13, fine, tWeldGun;
		MoveL [[1000.64,1624.71,1.80],[0.147993,-0.85301,-0.305288,-0.396575],[0,-1,-2,0],[9E+09,9E+09,9E+09,9E+09,9E+09,9E+09]], vmax, z50, tWeldGun;
		MoveJ [[999.85,699.71,74.25],[0.145952,0.855608,-0.347947,0.354353],[0,0,-2,0],[9E+09,9E+09,9E+09,9E+09,9E+09,9E+09]], vmax, z50, tWeldGun;
		MoveL [[1000.23,680.99,-33.60],[0.145957,0.855605,-0.347951,0.354355],[0,0,-2,0],[9E+09,9E+09,9E+09,9E+09,9E+09,9E+09]], vmax, z50, tWeldGun;
		ArcLStart [[1012.62,673.90,-46.78],[0.1719,0.826331,-0.335983,0.418023],[0,-1,-1,0],[9E+09,9E+09,9E+09,9E+09,9E+09,9E+09]], v10, seam13, weld13, fine, tWeldGun;
		ArcLEnd [[1014.09,670.24,-110.35],[0.203441,0.797575,-0.333295,0.459784],[0,-1,-1,0],[9E+09,9E+09,9E+09,9E+09,9E+09,9E+09]], v10, seam13, weld13, fine, tWeldGun;
		MoveL [[991.82,687.85,-113.61],[0.188232,0.8013,-0.32459,0.46597],[0,-1,-1,0],[9E+09,9E+09,9E+09,9E+09,9E+09,9E+09]], vmax, z50, tWeldGun;
		MoveL [[991.30,687.21,122.60],[0.188682,0.80133,-0.324494,0.465805],[0,-1,-1,0],[9E+09,9E+09,9E+09,9E+09,9E+09,9E+09]], vmax, z50, tWeldGun;
		MoveJ [[1353.61,686.57,-9.49],[0.257647,0.673939,-0.273385,0.636149],[0,-1,-1,0],[9E+09,9E+09,9E+09,9E+09,9E+09,9E+09]], vmax, z50, tWeldGun;
		MoveL [[1366.45,676.52,-47.24],[0.257646,0.673939,-0.273392,0.636147],[0,-1,-1,0],[9E+09,9E+09,9E+09,9E+09,9E+09,9E+09]], vmax, z50, tWeldGun;
		MoveL [[1385.74,669.35,-53.86],[0.230513,0.683708,-0.247774,0.646542],[0,-1,-1,0],[9E+09,9E+09,9E+09,9E+09,9E+09,9E+09]], vmax, z50, tWeldGun;
		ArcLStart [[1396.72,664.95,-53.87],[0.230521,0.683708,-0.247794,0.64653],[0,-1,-1,0],[9E+09,9E+09,9E+09,9E+09,9E+09,9E+09]], v10, seam13, weld13, fine, tWeldGun;
		ArcLEnd [[1395.51,665.99,-104.00],[0.221455,0.706537,-0.255943,0.621496],[0,-1,-1,0],[9E+09,9E+09,9E+09,9E+09,9E+09,9E+09]], v10, seam13, weld13, fine, tWeldGun;
		MoveL [[1331.35,694.89,21.64],[0.250476,0.690284,-0.28012,0.618307],[0,-1,-1,0],[9E+09,9E+09,9E+09,9E+09,9E+09,9E+09]], vmax, z50, tWeldGun;
		MoveJ [[1376.90,1623.22,41.45],[0.127213,-0.647245,-0.354873,-0.662538],[0,-1,-2,0],[9E+09,9E+09,9E+09,9E+09,9E+09,9E+09]], vmax, z50, tWeldGun;
		MoveL [[1376.90,1623.22,-50.53],[0.127212,-0.647239,-0.354892,-0.662534],[0,-1,-2,0],[9E+09,9E+09,9E+09,9E+09,9E+09,9E+09]], vmax, z50, tWeldGun;
		MoveL [[1397.45,1625.31,-50.53],[0.127209,-0.647235,-0.354904,-0.662533],[0,-1,-2,0],[9E+09,9E+09,9E+09,9E+09,9E+09,9E+09]], vmax, z50, tWeldGun;
		ArcLStart [[1408.53,1635.18,-50.45],[0.13106,-0.646617,-0.358565,-0.66041],[0,-1,-2,0],[9E+09,9E+09,9E+09,9E+09,9E+09,9E+09]], v10, seam13, weld13, fine, tWeldGun;
		ArcLEnd [[1408.03,1635.82,-99.67],[0.131146,-0.646603,-0.358564,-0.660407],[0,-1,-2,0],[9E+09,9E+09,9E+09,9E+09,9E+09,9E+09]], v10, seam13, weld13, fine, tWeldGun;
		MoveL [[1363.68,1613.53,-100.12],[0.126344,-0.650949,-0.356972,-0.657932],[0,-1,-2,0],[9E+09,9E+09,9E+09,9E+09,9E+09,9E+09]], vmax, z50, tWeldGun;
		MoveL [[1363.68,1613.52,239.17],[0.126341,-0.650966,-0.356946,-0.65793],[0,-1,-2,0],[9E+09,9E+09,9E+09,9E+09,9E+09,9E+09]], vmax, z50, tWeldGun;
		MoveJ [[1053.29,1631.94,67.33],[0.645571,-0.290399,-0.679976,-0.191155],[0,0,-4,0],[9E+09,9E+09,9E+09,9E+09,9E+09,9E+09]], vmax, z50, tWeldGun;
		MoveL [[1050.64,1634.55,-48.97],[0.636579,-0.309627,-0.673934,-0.211453],[0,0,-4,0],[9E+09,9E+09,9E+09,9E+09,9E+09,9E+09]], vmax, z50, tWeldGun;
		ArcLStart [[1024.87,1642.92,-50.56],[0.620533,-0.340261,-0.661431,-0.248335],[0,0,-4,0],[9E+09,9E+09,9E+09,9E+09,9E+09,9E+09]], v40, seam13, weld13, fine, tWeldGun;
		ArcLEnd [[1024.76,1640.88,-101.10],[0.608555,-0.344646,-0.672494,-0.242141],[0,0,-4,0],[9E+09,9E+09,9E+09,9E+09,9E+09,9E+09]], v10, seam13, weld13, fine, tWeldGun;
		MoveL [[1059.23,1614.28,-98.92],[0.62811,-0.294152,-0.696928,-0.18233],[0,0,-4,0],[9E+09,9E+09,9E+09,9E+09,9E+09,9E+09]], vmax, z50, tWeldGun;
		MoveL [[1059.23,1614.28,101.64],[0.628115,-0.294149,-0.696925,-0.182328],[0,0,-4,0],[9E+09,9E+09,9E+09,9E+09,9E+09,9E+09]], vmax, z50, tWeldGun;
		MoveJ [[1052.30,694.66,47.76],[0.644485,0.276131,-0.67942,0.216286],[0,-1,-5,0],[9E+09,9E+09,9E+09,9E+09,9E+09,9E+09]], vmax, z50, tWeldGun;
		MoveL [[1046.18,687.12,-54.58],[0.644485,0.276128,-0.679419,0.216291],[0,-1,-5,0],[9E+09,9E+09,9E+09,9E+09,9E+09,9E+09]], vmax, z50, tWeldGun;
		ArcLStart [[1016.59,670.93,-55.13],[0.641006,0.272426,-0.686489,0.208876],[0,-1,-5,0],[9E+09,9E+09,9E+09,9E+09,9E+09,9E+09]], v40, seam13, weld13, fine, tWeldGun;
		ArcLEnd [[1018.18,671.82,-104.69],[0.610333,0.278617,-0.715977,0.192985],[0,-1,-5,0],[9E+09,9E+09,9E+09,9E+09,9E+09,9E+09]], v10, seam13, weld13, fine, tWeldGun;
		MoveL [[1061.24,699.45,-98.70],[0.621239,0.282704,-0.701168,0.206166],[0,-1,-5,0],[9E+09,9E+09,9E+09,9E+09,9E+09,9E+09]], vmax, z50, tWeldGun;
		MoveL [[1054.68,728.71,93.69],[0.621244,0.28271,-0.701163,0.206161],[0,-1,-5,0],[9E+09,9E+09,9E+09,9E+09,9E+09,9E+09]], vmax, z50, tWeldGun;
		MoveJ pSafeS1, vmax, z50, tWeldGun;
	ENDPROC
	PROC ProSkid100()
		MoveJ [[1291.14,1401.40,237.11],[0.110665,-0.797291,0.0809156,-0.587821],[0,-1,-2,0],[9E+09,9E+09,9E+09,9E+09,9E+09,9E+09]], vmax, z50, tWeldGun;
		MoveL [[1375.22,1595.27,-52.82],[0.288027,-0.714876,-0.187844,-0.608858],[0,0,-3,0],[9E+09,9E+09,9E+09,9E+09,9E+09,9E+09]], vmax, z50, tWeldGun;
		ArcLStart [[1401.19,1605.13,-53.85],[0.288002,-0.715075,-0.187416,-0.608768],[0,0,-3,0],[9E+09,9E+09,9E+09,9E+09,9E+09,9E+09]], v40, seam13, weld13, fine, tWeldGun;
		ArcLEnd [[1398.73,1603.16,-97.27],[0.291491,-0.748178,-0.222798,-0.552834],[0,0,-3,0],[9E+09,9E+09,9E+09,9E+09,9E+09,9E+09]], v10, seam13, weld13, fine, tWeldGun;
		MoveL [[1364.33,1598.00,-103.67],[0.29149,-0.748144,-0.222826,-0.552868],[0,0,-3,0],[9E+09,9E+09,9E+09,9E+09,9E+09,9E+09]], vmax, z50, tWeldGun;
		MoveL [[1364.34,1597.99,108.74],[0.291485,-0.748128,-0.222876,-0.552873],[0,0,-3,0],[9E+09,9E+09,9E+09,9E+09,9E+09,9E+09]], vmax, z50, tWeldGun;
		MoveJ [[1362.85,671.57,209.86],[0.286582,0.681473,-0.261257,0.620653],[0,-1,-1,0],[9E+09,9E+09,9E+09,9E+09,9E+09,9E+09]], vmax, z50, tWeldGun;
		MoveL [[1362.83,671.44,-56.38],[0.286695,0.6814,-0.261216,0.620699],[0,-1,-1,0],[9E+09,9E+09,9E+09,9E+09,9E+09,9E+09]], vmax, z50, tWeldGun;
		ArcLStart [[1395.77,665.10,-57.82],[0.286611,0.681406,-0.26142,0.620645],[0,-1,-1,0],[9E+09,9E+09,9E+09,9E+09,9E+09,9E+09]], v40, seam13, weld13, fine, tWeldGun;
		ArcLEnd [[1394.43,667.22,-108.56],[0.265195,0.724641,-0.280093,0.571066],[0,-1,-1,0],[9E+09,9E+09,9E+09,9E+09,9E+09,9E+09]], v10, seam13, weld13, fine, tWeldGun;
		MoveL [[1359.52,678.30,-105.63],[0.265193,0.724636,-0.280059,0.57109],[0,-1,-1,0],[9E+09,9E+09,9E+09,9E+09,9E+09,9E+09]], vmax, z50, tWeldGun;
		MoveL [[1359.46,678.32,110.96],[0.265199,0.724649,-0.280131,0.571035],[0,-1,-1,0],[9E+09,9E+09,9E+09,9E+09,9E+09,9E+09]], vmax, z50, tWeldGun;
		MoveJ [[1044.44,682.04,140.05],[0.601349,0.276396,-0.690912,0.290906],[0,-1,-1,0],[9E+09,9E+09,9E+09,9E+09,9E+09,9E+09]], vmax, z50, tWeldGun;
		MoveL [[1044.44,682.04,-56.39],[0.601349,0.276385,-0.690916,0.290907],[0,-1,-1,0],[9E+09,9E+09,9E+09,9E+09,9E+09,9E+09]], vmax, z50, tWeldGun;
		ArcLStart [[1017.57,668.39,-58.10],[0.603558,0.271588,-0.6932,0.285364],[0,-1,-1,0],[9E+09,9E+09,9E+09,9E+09,9E+09,9E+09]], v40, seam13, weld13, fine, tWeldGun;
		ArcLEnd [[1019.45,669.58,-104.61],[0.590639,0.26522,-0.716441,0.259839],[0,-1,-1,0],[9E+09,9E+09,9E+09,9E+09,9E+09,9E+09]], v10, seam13, weld13, fine, tWeldGun;
		MoveL [[1053.53,682.10,-104.02],[0.581859,0.284263,-0.707585,0.282771],[0,-1,-1,0],[9E+09,9E+09,9E+09,9E+09,9E+09,9E+09]], vmax, z50, tWeldGun;
		MoveL [[1053.53,682.10,204.32],[0.581854,0.284262,-0.707586,0.282779],[0,-1,-1,0],[9E+09,9E+09,9E+09,9E+09,9E+09,9E+09]], vmax, z50, tWeldGun;
		MoveJ [[1060.34,1591.42,255.61],[0.587485,-0.309916,-0.701855,-0.25732],[0,0,0,0],[9E+09,9E+09,9E+09,9E+09,9E+09,9E+09]], vmax, z50, tWeldGun;
		MoveL [[1053.26,1597.30,-47.55],[0.593101,-0.251297,-0.715306,-0.270959],[0,0,0,0],[9E+09,9E+09,9E+09,9E+09,9E+09,9E+09]], vmax, z50, tWeldGun;
		ArcLStart [[1026.61,1608.02,-51.00],[0.610395,-0.281453,-0.687146,-0.275743],[0,0,0,0],[9E+09,9E+09,9E+09,9E+09,9E+09,9E+09]], v40, seam13, weld13, fine, tWeldGun;
		ArcLEnd [[1026.10,1606.98,-99.41],[0.589939,-0.305128,-0.703921,-0.251723],[0,0,0,0],[9E+09,9E+09,9E+09,9E+09,9E+09,9E+09]], v10, seam13, weld13, fine, tWeldGun;
		MoveL [[1060.35,1591.41,-99.10],[0.587476,-0.309917,-0.701859,-0.257327],[0,0,0,0],[9E+09,9E+09,9E+09,9E+09,9E+09,9E+09]], vmax, z50, tWeldGun;
		MoveL [[1060.34,1591.42,255.61],[0.587485,-0.309915,-0.701855,-0.25732],[0,0,0,0],[9E+09,9E+09,9E+09,9E+09,9E+09,9E+09]], vmax, z50, tWeldGun;
		SingArea\Wrist;
		MoveJ [[1013.97,1596.58,293.15],[0.294503,-0.721995,-0.258472,-0.57025],[0,-1,-2,0],[9E+09,9E+09,9E+09,9E+09,9E+09,9E+09]], vmax, z50, tWeldGun;
		MoveL [[1013.98,1596.59,-30.67],[0.294506,-0.721988,-0.258475,-0.570255],[0,-1,-2,0],[9E+09,9E+09,9E+09,9E+09,9E+09,9E+09]], vmax, z50, tWeldGun;
		ArcLStart [[1023.71,1603.83,-45.32],[0.294459,-0.722161,-0.258075,-0.570242],[0,-1,-2,0],[9E+09,9E+09,9E+09,9E+09,9E+09,9E+09]], v40, seam13, weld13, fine, tWeldGun;
		ArcLEnd [[1025.41,1604.13,-103.60],[0.29453,-0.721895,-0.258759,-0.570231],[0,-2,-1,0],[9E+09,9E+09,9E+09,9E+09,9E+09,9E+09]], v10, seam13, weld13, fine, tWeldGun;
		MoveL [[1013.24,1596.64,-103.54],[0.294541,-0.721861,-0.258796,-0.570252],[0,-2,-1,0],[9E+09,9E+09,9E+09,9E+09,9E+09,9E+09]], vmax, z50, tWeldGun;
		MoveL [[1013.24,1596.64,216.29],[0.294538,-0.721863,-0.258801,-0.570249],[0,-1,-2,0],[9E+09,9E+09,9E+09,9E+09,9E+09,9E+09]], vmax, z50, tWeldGun;
		MoveJ [[1006.20,679.01,292.67],[0.249851,0.680628,-0.312953,0.613499],[0,-1,-1,0],[9E+09,9E+09,9E+09,9E+09,9E+09,9E+09]], vmax, z50, tWeldGun;
		MoveL [[1006.17,679.00,-34.38],[0.24986,0.680635,-0.312969,0.61348],[0,-1,-1,0],[9E+09,9E+09,9E+09,9E+09,9E+09,9E+09]], vmax, z50, tWeldGun;
		ArcLStart [[1018.04,667.69,-51.11],[0.249871,0.680622,-0.312899,0.613525],[0,-1,-1,0],[9E+09,9E+09,9E+09,9E+09,9E+09,9E+09]], v40, seam13, weld13, fine, tWeldGun;
		ArcLEnd [[1018.17,669.74,-109.45],[0.216526,0.718194,-0.30883,0.584755],[0,-1,-1,0],[9E+09,9E+09,9E+09,9E+09,9E+09,9E+09]], v10, seam13, weld13, fine, tWeldGun;
		MoveL [[1006.90,676.88,-109.46],[0.216515,0.7182,-0.3088,0.584767],[0,-1,-1,0],[9E+09,9E+09,9E+09,9E+09,9E+09,9E+09]], vmax, z50, tWeldGun;
		MoveL [[1006.79,676.72,112.07],[0.216658,0.718018,-0.309197,0.584729],[0,-1,-1,0],[9E+09,9E+09,9E+09,9E+09,9E+09,9E+09]], vmax, z50, tWeldGun;
		MoveJ [[787.15,693.27,162.12],[0.200359,0.831329,-0.351726,0.38084],[0,-1,-1,0],[9E+09,9E+09,9E+09,9E+09,9E+09,9E+09]], vmax, z50, tWeldGun;
		MoveL [[803.22,683.52,-42.38],[0.200572,0.831304,-0.351703,0.380802],[0,-1,-1,0],[9E+09,9E+09,9E+09,9E+09,9E+09,9E+09]], vmax, z50, tWeldGun;
		ArcLStart [[820.10,672.81,-46.13],[0.200379,0.831311,-0.351741,0.380853],[0,-1,-1,0],[9E+09,9E+09,9E+09,9E+09,9E+09,9E+09]], v40, seam13, weld13, fine, tWeldGun;
		ArcL [[817.01,674.25,-61.57],[0.20037,0.83131,-0.351759,0.380844],[0,-1,-1,0],[9E+09,9E+09,9E+09,9E+09,9E+09,9E+09]], v5, seam13, weld13, z1, tWeldGun;
		ArcLEnd [[794.94,677.39,-61.37],[0.290522,0.768851,-0.506548,0.260529],[0,0,-1,0],[9E+09,9E+09,9E+09,9E+09,9E+09,9E+09]], v5, seam13, weld13, fine, tWeldGun;
		MoveL [[734.17,714.46,-10.08],[0.200543,0.831312,-0.351674,0.380825],[0,-1,-1,0],[9E+09,9E+09,9E+09,9E+09,9E+09,9E+09]], vmax, z50, tWeldGun;
		MoveJ [[728.25,1535.19,24.79],[0.147924,-0.86943,-0.34114,-0.325322],[0,0,-2,0],[9E+09,9E+09,9E+09,9E+09,9E+09,9E+09]], vmax, z50, tWeldGun;
		MoveL [[809.40,1591.07,-32.04],[0.147916,-0.869421,-0.341164,-0.325324],[0,0,-2,0],[9E+09,9E+09,9E+09,9E+09,9E+09,9E+09]], vmax, z50, tWeldGun;
		ArcLStart [[827.85,1598.76,-39.10],[0.147892,-0.869436,-0.341158,-0.325301],[0,0,-2,0],[9E+09,9E+09,9E+09,9E+09,9E+09,9E+09]], v40, seam13, weld13, fine, tWeldGun;
		ArcL [[824.60,1599.34,-54.56],[0.213243,-0.841559,-0.352486,-0.34937],[0,0,-2,0],[9E+09,9E+09,9E+09,9E+09,9E+09,9E+09]], v5, seam13, weld13, z1, tWeldGun;
		ArcLEnd [[804.61,1597.85,-55.38],[0.172397,-0.84314,-0.38332,-0.335351],[0,0,-2,0],[9E+09,9E+09,9E+09,9E+09,9E+09,9E+09]], v5, seam13, weld13, fine, tWeldGun;
		MoveL [[776.91,1584.46,5.55],[0.169992,-0.855201,-0.338248,-0.354009],[0,0,-2,0],[9E+09,9E+09,9E+09,9E+09,9E+09,9E+09]], vmax, z50, tWeldGun;
		MoveJ [[190.08,1566.54,31.00],[0.344053,-0.456867,-0.796918,-0.19448],[0,0,1,0],[9E+09,9E+09,9E+09,9E+09,9E+09,9E+09]], vmax, z50, tWeldGun;
		MoveL [[140.48,1600.64,-31.65],[0.344036,-0.456857,-0.79694,-0.194443],[0,0,1,0],[9E+09,9E+09,9E+09,9E+09,9E+09,9E+09]], vmax, z50, tWeldGun;
		ArcLStart [[132.97,1606.81,-38.27],[0.398419,-0.43769,-0.785543,-0.180589],[0,0,1,0],[9E+09,9E+09,9E+09,9E+09,9E+09,9E+09]], v40, seam13, weld13, fine, tWeldGun;
		ArcL [[137.87,1603.07,-53.48],[0.330333,-0.450337,-0.806737,-0.19301],[0,-1,1,0],[9E+09,9E+09,9E+09,9E+09,9E+09,9E+09]], v5, seam13, weld13, z1, tWeldGun;
		ArcLEnd [[160.89,1601.52,-53.60],[0.247106,-0.517365,-0.784142,-0.237474],[0,-1,1,0],[9E+09,9E+09,9E+09,9E+09,9E+09,9E+09]], v5, seam13, weld13, fine, tWeldGun;
		MoveL [[175.52,1584.51,-47.94],[0.344043,-0.456835,-0.796927,-0.194535],[0,0,1,0],[9E+09,9E+09,9E+09,9E+09,9E+09,9E+09]], vmax, z50, tWeldGun;
		MoveJ [[182.42,764.05,86.85],[0.357832,0.377008,-0.841375,0.14802],[0,0,0,0],[9E+09,9E+09,9E+09,9E+09,9E+09,9E+09]], vmax, z50, tWeldGun;
		MoveL [[138.47,690.39,-38.58],[0.357921,0.376925,-0.841359,0.148106],[0,0,0,0],[9E+09,9E+09,9E+09,9E+09,9E+09,9E+09]], vmax, z50, tWeldGun;
		ArcLStart [[127.27,682.76,-39.17],[0.357916,0.376949,-0.841354,0.148087],[0,0,0,0],[9E+09,9E+09,9E+09,9E+09,9E+09,9E+09]], v40, seam13, weld13, fine, tWeldGun;
		ArcL [[131.33,682.78,-57.87],[0.357887,0.376962,-0.841374,0.148009],[0,0,0,0],[9E+09,9E+09,9E+09,9E+09,9E+09,9E+09]], v5, seam13, weld13, z1, tWeldGun;
		ArcLEnd [[152.38,682.50,-58.95],[0.357948,0.376909,-0.841357,0.148091],[0,0,0,0],[9E+09,9E+09,9E+09,9E+09,9E+09,9E+09]], v5, seam13, weld13, fine, tWeldGun;
		MoveL [[182.36,703.78,23.74],[0.357926,0.376967,-0.841339,0.1481],[0,0,0,0],[9E+09,9E+09,9E+09,9E+09,9E+09,9E+09]], vmax, z50, tWeldGun;
		MoveJ [[104.88,808.11,108.60],[0.181133,-0.65989,-0.702536,-0.195398],[0,-1,1,0],[9E+09,9E+09,9E+09,9E+09,9E+09,9E+09]], vmax, z50, tWeldGun;
		MoveL [[104.87,808.11,-22.73],[0.181133,-0.6599,-0.702527,-0.195398],[0,-1,1,0],[9E+09,9E+09,9E+09,9E+09,9E+09,9E+09]], vmax, z50, tWeldGun;
		ArcLStart [[104.88,808.11,-33.52],[0.181134,-0.659877,-0.702547,-0.1954],[0,-1,1,0],[9E+09,9E+09,9E+09,9E+09,9E+09,9E+09]], v10, seam13, weld13, fine, tWeldGun;
		ArcLEnd [[119.95,808.11,-33.52],[0.181133,-0.659872,-0.702552,-0.195399],[0,-1,1,0],[9E+09,9E+09,9E+09,9E+09,9E+09,9E+09]], v10, seam13, weld13, fine, tWeldGun;
		MoveL [[119.95,808.11,110.38],[0.181135,-0.659885,-0.70254,-0.1954],[0,-1,1,0],[9E+09,9E+09,9E+09,9E+09,9E+09,9E+09]], vmax, z50, tWeldGun;
		MoveJ [[104.20,866.55,110.15],[0.247858,0.624252,-0.690017,0.269727],[0,-1,0,0],[9E+09,9E+09,9E+09,9E+09,9E+09,9E+09]], vmax, z50, tWeldGun;
		MoveL [[104.20,866.56,-18.99],[0.247849,0.624251,-0.690021,0.269728],[0,-1,0,0],[9E+09,9E+09,9E+09,9E+09,9E+09,9E+09]], vmax, z50, tWeldGun;
		ArcLStart [[104.22,866.56,-33.89],[0.247832,0.624264,-0.690012,0.269738],[0,-1,0,0],[9E+09,9E+09,9E+09,9E+09,9E+09,9E+09]], v10, seam13, weld13, fine, tWeldGun;
		ArcLEnd [[117.44,866.46,-33.99],[0.247835,0.624263,-0.690014,0.269732],[0,-1,0,0],[9E+09,9E+09,9E+09,9E+09,9E+09,9E+09]], v10, seam13, weld13, fine, tWeldGun;
		MoveL [[117.44,866.45,125.28],[0.247841,0.62426,-0.690014,0.269731],[0,-1,0,0],[9E+09,9E+09,9E+09,9E+09,9E+09,9E+09]], vmax, z50, tWeldGun;
		MoveJ [[108.37,1419.35,200.82],[0.287761,-0.638557,-0.653225,-0.28764],[0,-1,1,0],[9E+09,9E+09,9E+09,9E+09,9E+09,9E+09]], vmax, z50, tWeldGun;
		MoveL [[109.57,1420.53,-14.32],[0.263504,-0.648771,-0.662871,-0.265072],[0,-1,1,0],[9E+09,9E+09,9E+09,9E+09,9E+09,9E+09]], vmax, z50, tWeldGun;
		ArcLStart [[109.57,1420.55,-29.31],[0.263511,-0.648758,-0.662878,-0.26508],[0,-1,1,0],[9E+09,9E+09,9E+09,9E+09,9E+09,9E+09]], v10, seam13, weld13, fine, tWeldGun;
		ArcLEnd [[121.97,1420.55,-29.31],[0.26351,-0.648759,-0.662878,-0.265081],[0,-1,1,0],[9E+09,9E+09,9E+09,9E+09,9E+09,9E+09]], v10, seam13, weld13, fine, tWeldGun;
		MoveL [[121.96,1420.55,113.82],[0.263512,-0.648767,-0.662871,-0.265077],[0,-1,1,0],[9E+09,9E+09,9E+09,9E+09,9E+09,9E+09]], vmax, z50, tWeldGun;
		MoveJ [[107.74,1476.86,132.75],[0.227381,0.67854,-0.65675,0.237825],[0,0,-1,0],[9E+09,9E+09,9E+09,9E+09,9E+09,9E+09]], vmax, z50, tWeldGun;
		MoveL [[107.75,1476.86,-6.53],[0.227369,0.678545,-0.656746,0.237835],[0,0,-1,0],[9E+09,9E+09,9E+09,9E+09,9E+09,9E+09]], vmax, z50, tWeldGun;
		ArcLStart [[105.63,1476.40,-27.57],[0.227388,0.678538,-0.656756,0.237808],[0,0,-1,0],[9E+09,9E+09,9E+09,9E+09,9E+09,9E+09]], v40, seam13, weld13, fine, tWeldGun;
		ArcLEnd [[119.62,1476.10,-27.13],[0.227387,0.678539,-0.656755,0.237809],[0,0,-1,0],[9E+09,9E+09,9E+09,9E+09,9E+09,9E+09]], v10, seam13, weld13, fine, tWeldGun;
		MoveL [[118.38,1476.85,2.29],[0.227385,0.678544,-0.656744,0.237828],[0,0,-1,0],[9E+09,9E+09,9E+09,9E+09,9E+09,9E+09]], vmax, z50, tWeldGun;
		MoveL [[836.49,1471.77,-21.22],[0.227415,0.678515,-0.656775,0.237796],[0,0,-1,0],[9E+09,9E+09,9E+09,9E+09,9E+09,9E+09]], vmax, z50, tWeldGun;
		ArcLStart [[833.70,1470.86,-31.25],[0.227422,0.678532,-0.656755,0.237797],[0,0,-1,0],[9E+09,9E+09,9E+09,9E+09,9E+09,9E+09]], v10, seam13, weld13, fine, tWeldGun;
		ArcLEnd [[848.24,1470.72,-30.35],[0.227417,0.67853,-0.656757,0.2378],[0,0,-1,0],[9E+09,9E+09,9E+09,9E+09,9E+09,9E+09]], v10, seam13, weld13, fine, tWeldGun;
		MoveL [[845.94,1471.75,199.33],[0.227429,0.678527,-0.65675,0.237818],[0,0,-1,0],[9E+09,9E+09,9E+09,9E+09,9E+09,9E+09]], vmax, z50, tWeldGun;
		MoveJ [[851.82,1398.82,138.77],[0.249585,-0.660425,-0.662158,-0.251183],[0,-1,1,0],[9E+09,9E+09,9E+09,9E+09,9E+09,9E+09]], vmax, z50, tWeldGun;
		MoveL [[851.80,1413.16,-17.04],[0.24959,-0.660434,-0.662152,-0.251173],[0,-1,1,0],[9E+09,9E+09,9E+09,9E+09,9E+09,9E+09]], vmax, z50, tWeldGun;
		ArcLStart [[851.81,1413.17,-30.35],[0.249586,-0.660427,-0.662156,-0.251181],[0,-1,1,0],[9E+09,9E+09,9E+09,9E+09,9E+09,9E+09]], v40, seam13, weld13, fine, tWeldGun;
		ArcLEnd [[837.71,1413.17,-30.35],[0.249589,-0.660431,-0.662154,-0.251176],[0,-1,1,0],[9E+09,9E+09,9E+09,9E+09,9E+09,9E+09]], v10, seam13, weld13, fine, tWeldGun;
		MoveL [[837.70,1413.16,114.72],[0.24959,-0.660435,-0.662151,-0.251172],[0,-1,1,0],[9E+09,9E+09,9E+09,9E+09,9E+09,9E+09]], vmax, z50, tWeldGun;
		MoveJ [[836.86,863.49,66.47],[0.245499,0.671633,-0.652073,0.251873],[0,0,-1,0],[9E+09,9E+09,9E+09,9E+09,9E+09,9E+09]], vmax, z50, tWeldGun;
		MoveL [[833.18,862.81,-20.93],[0.245535,0.671618,-0.652081,0.251858],[0,0,-1,0],[9E+09,9E+09,9E+09,9E+09,9E+09,9E+09]], vmax, z50, tWeldGun;
		ArcLStart [[832.14,861.68,-36.34],[0.245527,0.671615,-0.652094,0.25184],[0,0,-1,0],[9E+09,9E+09,9E+09,9E+09,9E+09,9E+09]], v40, seam13, weld13, fine, tWeldGun;
		ArcLEnd [[847.39,860.80,-37.23],[0.245547,0.671614,-0.652088,0.251841],[0,0,-1,0],[9E+09,9E+09,9E+09,9E+09,9E+09,9E+09]], v10, seam13, weld13, fine, tWeldGun;
		MoveL [[844.19,862.64,90.70],[0.24553,0.671618,-0.652082,0.251861],[0,0,-1,0],[9E+09,9E+09,9E+09,9E+09,9E+09,9E+09]], vmax, z50, tWeldGun;
		MoveJ [[850.02,796.71,104.60],[0.232706,-0.667694,-0.66755,-0.23326],[0,-1,1,0],[9E+09,9E+09,9E+09,9E+09,9E+09,9E+09]], vmax, z50, tWeldGun;
		MoveL [[848.57,804.07,-20.25],[0.232717,-0.667711,-0.667535,-0.233244],[0,-1,1,0],[9E+09,9E+09,9E+09,9E+09,9E+09,9E+09]], vmax, z50, tWeldGun;
		ArcLStart [[848.57,804.08,-35.68],[0.232715,-0.667709,-0.667535,-0.233251],[0,-1,1,0],[9E+09,9E+09,9E+09,9E+09,9E+09,9E+09]], v40, seam13, weld13, fine, tWeldGun;
		ArcLEnd [[836.56,803.94,-35.91],[0.232718,-0.667714,-0.66753,-0.233248],[0,-1,1,0],[9E+09,9E+09,9E+09,9E+09,9E+09,9E+09]], v10, seam13, weld13, fine, tWeldGun;
		MoveL [[836.55,803.93,282.92],[0.232721,-0.66772,-0.667527,-0.233237],[0,-1,1,0],[9E+09,9E+09,9E+09,9E+09,9E+09,9E+09]], vmax, z50, tWeldGun;
		MoveJ pSafeS1, vmax, z50, tWeldGun;
	ENDPROC
ENDMODULE
